(* Prozess Stop *)
IF RisingEdgeProcessStop.Q THEN
	IF NOT(T_Process.T_Ctrle.xDone) AND NOT(T_Process.T_Fct.xExecute) THEN
		(* Prozess muss Aktiv sein und dürfte auch im ZyklusStop Zustand sein, welches dann unterbrochen werden würde *)
		T_Process.T_Fct.xStop:=T_Process.T_Ctrle.xStop;
	ELSE
		T_Process.T_Ctrle.xStop:=FALSE;
	END_IF;
END_IF;
(* Abbrechen des Prozesses *)
IF RisingEdgeProcessAbord.Q THEN
	T_Process.T_Fct.xAbordProcess:=TRUE;
END_IF;
(* Auffangen des Prozess Endes *)
IF NOT(T_Process.T_Ctrle.xDone) AND NOT(T_Process.T_Ctrle.xErrorReady) THEN
	IF NOT(T_Process.T_Fct.xExecute) AND T_Process.T_Fct.xDone THEN
		xSetEnd:=TRUE;
	END_IF;
END_IF;
END_ACTION
ACTION CtrlWorkpiece:
RisingEdgeCheckWorkEnd(CLK:=TStation_Work_St1.THWWorkStation.TCtrlWork.xWorkingFinished);
IF RisingEdgeCheckWorkEnd.Q AND xAutoActiveProcess AND (TStation_Work_St1.THWWorkStation.TCtrlWork.bPartQuality <> 0) AND
     (TStation_Work_St1.THWWorkStation.TCtrlWork.bPartQuality <> 7) AND (TStation_Work_St1.THWWorkStation.TCtrlWork.bPartQuality <> 8) THEN
	(* Nach jeder bearbeitenden Bohrung muss "xAddToolCounter_Machine" gesetzt werden-->Ist für den WzWechsel *)
	TStation_Work_St1.THWWorkStation.TCtrlWork.xAddToolCounter_Machine:=TRUE;
END_IF;
IF xHoleToWork THEN
	IF NOT(xWriteData) THEN
		IF (T_NovRam.T_Parameter.T_PartAnalysis[gciStationSt1].diActual_NumberHoleToWork <= 0) THEN
			T_NovRam.T_Parameter.T_PartAnalysis[gciStationSt1].diActual_NumberHoleToWork:=1;
		END_IF;
		FOR ii:= 1 TO ciMaxWP DO
			IF (T_NovRam.T_Parameter.T_PartAnalysis[gciStationSt1].adiNumberHole[ii] = T_NovRam.T_Parameter.T_PartAnalysis[gciStationSt1].diActual_NumberHoleToWork) THEN
				IF ((T_NovRam.T_Parameter.T_PartAnalysis[gciStationSt1].abWorkPartQuality[ii] >= 1) AND (T_NovRam.T_Parameter.T_PartAnalysis[gciStationSt1].abWorkPartQuality[ii] <= 6)) OR (T_NovRam.T_Parameter.T_PartAnalysis[gciStationSt1].abWorkPartQuality[ii] = 10) THEN
					T_NovRam.T_Parameter.T_PartAnalysis[gciStationSt1].diActual_NumberHoleToWork:=T_NovRam.T_Parameter.T_PartAnalysis[gciStationSt1].diActual_NumberHoleToWork + 1;
				END_IF;
			END_IF;
		END_FOR;
		(* Überprüfe ob Arrayelement erreicht wurde *)
		IF (T_NovRam.T_Parameter.T_PartAnalysis[gciStationSt1].diActual_NumberHoleToWork > T_NovRam.T_Parameter.T_PartAnalysis[gciStationSt1].adiNumberHole[ciMaxWP]) THEN
			FOR ii:=1 TO (ciMaxWP-1) DO
				T_NovRam.T_Parameter.T_PartAnalysis[gciStationSt1].abWorkPartQuality[ii]:=T_NovRam.T_Parameter.T_PartAnalysis[gciStationSt1].abWorkPartQuality[ii+1];
				T_NovRam.T_Parameter.T_PartAnalysis[gciStationSt1].arFirstHC[ii]:=T_NovRam.T_Parameter.T_PartAnalysis[gciStationSt1].arFirstHC[ii+1];
				T_NovRam.T_Parameter.T_PartAnalysis[gciStationSt1].aiHCCounter[ii]:=T_NovRam.T_Parameter.T_PartAnalysis[gciStationSt1].aiHCCounter[ii+1];
				T_NovRam.T_Parameter.T_PartAnalysis[gciStationSt1].aiHCCounterCentering[ii]:=T_NovRam.T_Parameter.T_PartAnalysis[gciStationSt1].aiHCCounterCentering[ii+1];
				T_NovRam.T_Parameter.T_PartAnalysis[gciStationSt1].aiHCCounterTorque[ii]:=T_NovRam.T_Parameter.T_PartAnalysis[gciStationSt1].aiHCCounterTorque[ii+1];
				T_NovRam.T_Parameter.T_PartAnalysis[gciStationSt1].aiHCCounterSpeed[ii]:=T_NovRam.T_Parameter.T_PartAnalysis[gciStationSt1].aiHCCounterSpeed[ii+1];
				T_NovRam.T_Parameter.T_PartAnalysis[gciStationSt1].adiCycleTime[ii]:=T_NovRam.T_Parameter.T_PartAnalysis[gciStationSt1].adiCycleTime[ii+1];
				T_NovRam.T_Parameter.T_PartAnalysis[gciStationSt1].adiWorkTime[ii]:=T_NovRam.T_Parameter.T_PartAnalysis[gciStationSt1].adiWorkTime[ii+1];
				T_NovRam.T_Parameter.T_PartAnalysis[gciStationSt1].abInfeedCounterZ[ii]:=T_NovRam.T_Parameter.T_PartAnalysis[gciStationSt1].abInfeedCounterZ[ii+1];
				T_NovRam.T_Parameter.T_PartAnalysis[gciStationSt1].adiNumberHole[ii]:=T_NovRam.T_Parameter.T_PartAnalysis[gciStationSt1].adiNumberHole[ii+1];
			END_FOR;
			T_NovRam.T_Parameter.T_PartAnalysis[gciStationSt1].abWorkPartQuality[ciMaxWP]:=0;
			T_NovRam.T_Parameter.T_PartAnalysis[gciStationSt1].arFirstHC[ciMaxWP]:=0.0;
			T_NovRam.T_Parameter.T_PartAnalysis[gciStationSt1].aiHCCounter[ciMaxWP]:=0;
			T_NovRam.T_Parameter.T_PartAnalysis[gciStationSt1].aiHCCounterCentering[ciMaxWP]:=0;
			T_NovRam.T_Parameter.T_PartAnalysis[gciStationSt1].aiHCCounterTorque[ciMaxWP]:=0;
			T_NovRam.T_Parameter.T_PartAnalysis[gciStationSt1].aiHCCounterSpeed[ciMaxWP]:=0;
			T_NovRam.T_Parameter.T_PartAnalysis[gciStationSt1].adiCycleTime[ciMaxWP]:=0;
			T_NovRam.T_Parameter.T_PartAnalysis[gciStationSt1].adiWorkTime[ciMaxWP]:=0;
			T_NovRam.T_Parameter.T_PartAnalysis[gciStationSt1].abInfeedCounterZ[ciMaxWP]:=0;
			T_NovRam.T_Parameter.T_PartAnalysis[gciStationSt1].adiNumberHole[ciMaxWP]:=T_NovRam.T_Parameter.T_PartAnalysis[gciStationSt1].adiNumberHole[ciMaxWP] + 1;
		END_IF;
		xHoleToWork:=FALSE;
	END_IF;
END_IF;
END_ACTION
ACTION ProcessFunction_Ctrl_End:
IF T_Process.T_Fct.xSetEndFunction OR xPrcFct_ForceResetFlag THEN
	IF NOT(xPrcFct_ForceResetFlag) THEN
		T_Process.T_Fct.xDone:=TRUE;
	END_IF;
	xPrcFct_ForceResetFlag:=FALSE;
	T_Process.T_Fct.xStop:=FALSE;
	T_Process.T_Fct.xExecute:=FALSE;
	T_Process.T_Fct.xAbordProcess:=FALSE;
	T_Process.T_Fct.xError:=FALSE;
	T_Process.T_Fct.diErrorNr:=0;
	T_Process.T_Fct.xQuitError:=FALSE;
	T_Process.T_Fct.xSetEndFunction:=FALSE;
	T_Process.T_Fct.xReset:=FALSE;
	xPrcFct_SaveStationError:=FALSE;
	xPrcFct_StartPrc_Parallel1:=FALSE;
	xPrcFct_StartPrc_Parallel2:=FALSE;
	iPrcFct_StepPrc_Parallel1:=1;
	iPrcFct_StepPrc_Parallel2:=1;
	xPrcFct_InitStep_Parallel1:=FALSE;
	xPrcFct_InitStep_Parallel2:=FALSE;
	xPrcFct_SetNextStationActive_St1:=FALSE;
	iPrcFct_PickPlaceProcedure:=0;
	xPrcFct_PartDiscReady:=FALSE;
	xPrcFct_ReadyToWriteQuality_St1:=FALSE;
	xPrcFct_XAxisGoToWaitPos:=FALSE;
	xPrcFct_ProcessContinueActive:=FALSE;
	iPrcFct_StepPrc:=1;
	xPrcFct_InitStep:=FALSE;
	xPrcFct_SaveNoMoreParts:=FALSE;
	xPrcFct_StopProcess:=FALSE;
	xPrcFct_StopCycleProcess:=FALSE;
	diPrcFct_SaveErrorNr:=0;
	TStation_Work.THWWorkStation.TCtrlWork.xWP_Analyse_ActiveCycle:=FALSE;			(* Zykluszeit für zu bearbeitende Bohrung ist gestartet *)
	TStation_Work.THWWorkStation.TCtrlWork.xWP_Analyse_ActiveWork:=FALSE;			(* Bearbeitungszeit für zu bearbeitende Bohrung ist gestartet *)
	xStartWorkPart:=FALSE;
	QxCoolant_St1:=FALSE;
	QxFastStrokeOn_St1:=FALSE;
END_IF;
END_ACTION
ACTION ProcessFunction_Ctrl_Error:
xPrcFct_StationError:=	TStation_Work.TControl.xError OR T_ProcessData.T_Ctrle.xErr;
IF (xPrcFct_StationError OR xPrcFct_SaveStationError) AND NOT(T_Process.T_Fct.xErrorReady) THEN
	xPrcFct_SaveStationError:=TRUE;
	IF (T_Process.T_Fct.iFunctNr = 2) THEN
		(* Automat *)
		xPrcFct_WorkStationReady:=	TStation_Work.TControl.xError OR NOT(xStartWorkPart);
	ELSE
		(* Restliche Prozesse *)
		xPrcFct_WorkStationReady:=	(TStation_Work.TControl.xError OR TStation_Work.TControl.xDone);
	END_IF;
	xPrcFct_StationReady:=	(xPrcFct_WorkStationReady OR xPrcFct_StationBlock);
	CASE iPrcFct_StepStationError OF
	(* Abwarten bis alle Station Zyklus beendet haben *)
	1: 	IF xPrcFct_StationReady THEN
			xPrcFct_StationBlock:=TRUE;
			iPrcFct_StepStationError:=iPrcFct_StepStationError + 1;
			IF TStation_Work.THWWorkStation.TCtrlWork.xWorkStartToolRotation THEN
				TStation_Work.THWWorkStation.TCtrlWork.xWorkStopToolRotation:=TRUE;
			END_IF;
		END_IF;
	2:	iPrcFct_StepStationError:=iPrcFct_StepStationError + 1;
		TStation_Work.THWWorkStation.TCtrlWork.xActiveProcess:=FALSE;
		TStation_Work.THWWorkStation.TCtrlWork.xWorkingFinished:=FALSE;
	(* Überprüfen ob es einen Fehler oder eine Warnung ist *)
	3:	IF (diPrcFct_SaveErrorNr <> 0)THEN
			T_Process.T_Fct.diErrorNr:=diPrcFct_SaveErrorNr;
		ELSIF TStation_Work.TControl.xError THEN
			T_Process.T_Fct.diErrorNr:=TStation_Work.TControl.diErrorNr;
		ELSIF T_ProcessData.T_Ctrle.xErr THEN
			T_Process.T_Fct.diErrorNr:=82000000 + T_ProcessData.T_Ctrle.udiErrorID;
		END_IF;
		FBErrorMessage(	diErrorNr:=T_Process.T_Fct.diErrorNr,
							T_ErrorList:=T_ErrorList);
		T_Process.T_Fct.xError:=TRUE;
		diPrcFct_SaveErrorNr:=0;
		iPrcFct_StepStationError:=iPrcFct_StepStationError + 1;
	(* Warten bis Quittiert wird *)
	4:	IF T_Process.T_Fct.xQuitError THEN
			T_Process.T_Fct.xQuitError:=FALSE;
			T_Process.T_Fct.xErrorReady:=TRUE;
			T_Process.T_Fct.xError:=FALSE;
			T_Process.T_Fct.xSetEndFunction:=TRUE;
		END_IF;
	END_CASE;
ELSE
	xExecuteOneTime:=FALSE;
	iPrcFct_StepStationError:=1;
END_IF;
END_ACTION
ACTION ProcessFunction_Ctrl_Main:
(* Prozess Start *)
IF T_Process.T_Fct.xExecute THEN
	T_Process.T_Fct.xStop:=FALSE;
	T_Process.T_Fct.xExecute:=FALSE;
	T_Process.T_Fct.xDone:=FALSE;
	T_Process.T_Fct.xAbordProcess:=FALSE;
	T_Process.T_Fct.xError:=FALSE;
	T_Process.T_Fct.diErrorNr:=0;
	iPrcFct_StepPrc:=1;
	xPrcFct_InitStep:=FALSE;
	xPrcFct_StartMainPrc:=TRUE;
	diPrcFct_SaveErrorNr:=0;
	TStation_Work.THWWorkStation.TCtrlWork.xWorkStartToolRotation:=FALSE;
	TStation_Work.THWWorkStation.TCtrlWork.xWorkStopToolRotation:=FALSE;
	TStation_Work.THWWorkStation.TCtrlWork.xWorkingFinished:=FALSE;
	xPrcFct_SaveNoMoreParts:=FALSE;
	xProcessActive:=FALSE;
END_IF;
(* Abbrechen des Prozesses *)
IF T_Process.T_Fct.xAbordProcess THEN
	T_Process.T_Fct.xAbordProcess:=FALSE;
	T_Process.T_Fct.xSetEndFunction:=TRUE;
END_IF;
IF NOT(xPrcFct_ForceResetFlag) AND xPrcFct_ProcessContinueActive THEN
	xPrcFct_StationBlock:=FALSE;
END_IF;
END_ACTION
ACTION ProcessFunction_Ctrl_Reset:
IF T_Process.T_Fct.xReset THEN
	T_Process.T_Fct.xSetEndFunction:=TRUE;
END_IF;
END_ACTION
ACTION ProcessFunction_Ctrl_Stop:
IF T_Process.T_Fct.xStop OR xPrcFct_StopProcess THEN
	xPrcFct_StationReady:=	NOT(TStation_Work.TControl.xExecute) AND (TStation_Work.TControl.xDone OR TStation_Work.TControl.xError);
	CASE iPrcFct_StepStopProcess OF
	(* Stoppen der Aktiven Stationen *)
	1:	xPrcFct_StationBlock:=TRUE;
		xPrcFct_StopProcess:=TRUE;
		xPrcFct_ProcessContinueActive:=FALSE;
		TStation_Work.TControl.xStop:=NOT(TStation_Work.TControl.xError) AND NOT(TStation_Work.TControl.xDone) AND xEnergyON;
		(* Flag für die WstkAnalyse zurücksetzen *)
		iPrcFct_StepStopProcess:=iPrcFct_StepStopProcess + 1;
	(* Zurücksetzen der Steuerflag für Bearbstationen *)
	2:	IF xPrcFct_StationReady OR xPrcFct_SaveStationError THEN
			iPrcFct_StepStopProcess:=iPrcFct_StepStopProcess + 1;
			TStation_Work.THWWorkStation.TCtrlWork.xActiveProcess:=FALSE;
			TStation_Work.THWWorkStation.TCtrlWork.xWorkingFinished:=FALSE;
			TStation_Work.THWWorkStation.TCtrlWork.xWorkStopToolRotation:=xEnergyON;
			(* Flag für die WstkAnalyse zurücksetzen *)
		END_IF;
	3:	IF (T_Process.T_Ctrle.iFunctNr <> 1) THEN
			TStation_Work.TControl.iFunctNr:=2;			(* Bearbeitungsstation Grundstellung *)
			TStation_Work.TControl.xExecute:=NOT(TStation_Work.TControl.xError) AND xEnergyON;
			IF (TStation_Work.THWWorkStation.TCtrlWork.bPartQuality >= 1) AND (TStation_Work.THWWorkStation.TCtrlWork.bPartQuality <= 6) THEN
				IF T_NovRam.T_Parameter.T_Machine.T_ParamSystem.xDataFileActive AND NOT(T_NovRam.T_Parameter.T_Machine.xEndlessProcessActive) THEN
					(* Prozessdatei wird geschrieben *)
					T_ProcessData.T_Ctrle.iFunction:=1;
					T_ProcessData.T_Ctrle.xExecute:=TRUE;
				END_IF;
			END_IF;
		END_IF;
		iPrcFct_StepStopProcess:=iPrcFct_StepStopProcess + 1;
	4:	IF NOT(TStation_Work.TControl.xExecute) AND (TStation_Work.TControl.xDone OR TStation_Work.TControl.xError) THEN
			iPrcFct_StepStopProcess:=iPrcFct_StepStopProcess + 1;
		END_IF;
	(* Abwarten bis alle Stationen bereit stehen *)
	5:	IF xPrcFct_StationReady OR xPrcFct_SaveStationError THEN
			iPrcFct_StepStopProcess:=iPrcFct_StepStopProcess + 1;
		END_IF;
	6:	xPrcFct_StopProcess:=FALSE;
		T_Process.T_Fct.xStop:=FALSE;
		IF NOT(xPrcFct_SaveStationError) THEN
			T_Process.T_Fct.xAbordProcess:=TRUE;
		END_IF;
	END_CASE;
ELSE
	iPrcFct_StepStopProcess:=1;
END_IF;
END_ACTION
ACTION ProcessFunction_Fct_Automat:
(******************************************************************************************************************************************)
(****************************				           Reset Processfunktion                                            *****************************)
(******************************************************************************************************************************************)
ProcessFunction_Ctrl_Reset;
(******************************************************************************************************************************************)
(****************************			        Processfunktion Fehler Controller                                    *****************************)
(******************************************************************************************************************************************)
ProcessFunction_Ctrl_Error;
(******************************************************************************************************************************************)
(****************************				    Processfunktion Haupt Controller                               *****************************)
(******************************************************************************************************************************************)
ProcessFunction_Ctrl_Main;
(******************************************************************************************************************************************)
(****************************			         Processfunktion sofort Unterbrechung                           *****************************)
(******************************************************************************************************************************************)
ProcessFunction_Ctrl_Stop;
(******************************************************************************************************************************************)
(****************************			             Processfunktion Hauptablauf                                       *****************************)
(******************************************************************************************************************************************)
ProcessFunction_Fct_Automat_Station;
IF xPrcFct_StartMainPrc AND NOT(xPrcFct_StationBlock) AND NOT(T_Process.T_Fct.xSetEndFunction) AND NOT(xPrcFct_SaveStationError) THEN
	CASE iPrcFct_StepPrc OF
	1:	T_ExchgParam.T_Visu.T_Message.iState:=0;
		IF (T_NovRam.T_Parameter.T_StationWork[gciStationSt1].T_ToolCounter.diMaxNumberToolCycle <> 0) AND
		    (T_NovRam.T_Parameter.T_StationWork[gciStationSt1].T_ToolCounter.diToolCycleCounter >= T_NovRam.T_Parameter.T_StationWork[gciStationSt1].T_ToolCounter.diMaxNumberToolCycle) THEN
			TStation_Work.TControl.xError:=TRUE;
			TStation_Work.TControl.xDone:=FALSE;
			TStation_Work.TControl.diErrorNr:=(gciStationSt1 * 1000000) + 16#F101;		(* WzWechsel muss vorgenommen werden *)
			RETURN;
		END_IF;
		IF (garPositionEndProcCalc[1] > T_NovRam.T_Parameter.T_StationWork[gciStationSt1].T_StProcess.rPositionEndProcMaxInc) AND (T_NovRam.T_Parameter.T_StationWork[gciStationSt1].T_StProcess.xPositionEndProcIncOnOff OR gxProcessCylindricalAreaActive) THEN
			TStation_Work.TControl.xError:=TRUE;
			TStation_Work.TControl.xDone:=FALSE;
			TStation_Work.TControl.diErrorNr:=(gciStationSt1 * 1000000) + 17;		(* Z Bearb EndPos Berechn. > Z Bearb EndPos Max *)
			RETURN;
		END_IF;
		IF (garCentringEndProcCalc[1] > T_NovRam.T_Parameter.T_StationWork[gciStationSt1].T_StProcess.rPositionEndProcMaxInc) AND T_NovRam.T_Parameter.T_StationWork[gciStationSt1].T_StProcess.xCentringEndProcIncOnOff THEN
			TStation_Work.TControl.xError:=TRUE;
			TStation_Work.TControl.xDone:=FALSE;
			TStation_Work.TControl.diErrorNr:=(gciStationSt1 * 1000000) + 19;		(* Z ZentrierPos berechn. > Z Bearb EndPos Max *)
			RETURN;
		END_IF;
		IF NOT(xPrcFct_InitStep) THEN
			xPrcFct_InitStep:=TRUE;
			gdiSavePartQuality:=0;
			xHoleToWork:=TRUE;
		END_IF;
		IF NOT(xHoleToWork) THEN
			xPrcFct_InitStep:=FALSE;
			iPrcFct_StepPrc:=iPrcFct_StepPrc + 1;
		END_IF;
	2:	IF NOT(xPrcFct_InitStep) THEN
			xPrcFct_InitStep:=TRUE;
			TStation_Work.TControl.iFunctNr:=2;		(* Bearbeitungsstation Grundstellung *)
			TStation_Work.TControl.xExecute:=TRUE;
			TStation_Work.THWWorkStation.TCtrlWork.xWP_Analyse_ActiveCycle:=TRUE;			(* Zykluszeit für zu bearbeitende Bohrung ist gestartet *)
		END_IF;
		IF NOT(TStation_Work.TControl.xExecute) AND TStation_Work.TControl.xDone THEN
			TStation_Work.THWWorkStation.TCtrlWork.xWorkStartToolRotation:=TRUE;
			xPrcFct_InitStep:=FALSE;
			iPrcFct_StepPrc:=iPrcFct_StepPrc + 1;
		END_IF;
	3:	IF NOT(xPrcFct_InitStep) THEN
			xPrcFct_InitStep:=TRUE;
			xStartWorkPart:=TRUE;
		END_IF;
		IF NOT(xStartWorkPart) THEN
			xPrcFct_InitStep:=FALSE;
			iPrcFct_StepPrc:=90;
		END_IF;
	90:	iPrcFct_StepPrc:=1;
		xPrcFct_InitStep:=FALSE;
		IF NOT(T_NovRam.T_Parameter.T_Machine.xEndlessProcessActive) THEN
			xPrcFct_StartMainPrc:=FALSE;
			T_Process.T_Fct.xSetEndFunction:=TRUE;	(* Prozess beendet *)
		END_IF;
	END_CASE;
END_IF;
(******************************************************************************************************************************************)
(****************************			             Processfunktion Parallelablauf                                       *****************************)
(******************************************************************************************************************************************)
IF NOT(xPrcFct_StationBlock) AND NOT(T_Process.T_Fct.xSetEndFunction) AND NOT(xPrcFct_SaveStationError) THEN
	IF xPrcFct_StartPrc_Parallel1 THEN
		CASE iPrcFct_StepPrc_Parallel1 OF
		1:	iPrcFct_StepPrc_Parallel1:=1;
			xPrcFct_InitStep_Parallel1:=FALSE;
			xPrcFct_StartPrc_Parallel1:=FALSE;
		END_CASE;
	END_IF;
	IF xPrcFct_StartPrc_Parallel2 THEN
		CASE iPrcFct_StepPrc_Parallel2 OF
		1:	iPrcFct_StepPrc_Parallel2:=1;
			xPrcFct_InitStep_Parallel2:=FALSE;
			xPrcFct_StartPrc_Parallel2:=FALSE;
		END_CASE;
	END_IF;
END_IF;
(******************************************************************************************************************************************)
(****************************				     Processfunktion Endprozedur                                    *****************************)
(******************************************************************************************************************************************)
ProcessFunction_Ctrl_End;
END_ACTION
ACTION ProcessFunction_Fct_Automat_Station:
(*********************************************************************************************************************************)
(***********************************			BEARBSTATION RECHTS			***********************************)
(*********************************************************************************************************************************)
IF xStartWorkPart AND NOT(xPrcFct_StationBlock) THEN
	CASE iStepPrc_1 OF
	(* Zuerst überprüfen welche WstkNummer bearbeitet werden muss *)
	1:	iStepPrc_1:=iStepPrc_1 + 1;
		xInitPrc_1:=FALSE;
		xBlockQuality_StR:=FALSE;
		iNumberTryInfeed:=0;
		TStation_Work.THWWorkStation.TCtrlWork.xLastTryInfeed:=FALSE;
	(* .StationFunction_Fct_04_InfeedWorking*)
	2:	IF NOT(xInitPrc_1) THEN
			xInitPrc_1:=TRUE;
			TStation_Work.TControl.iFunctNr:=4;			(* Wz in das Wstk einfädeln *)
			TStation_Work.TControl.xExecute:=TRUE;
			gxSuspensionONOFF:=TRUE;
		END_IF;
		IF NOT(TStation_Work.TControl.xExecute) AND TStation_Work.TControl.xDone THEN
			gxAddInfeedZ:=TRUE;
			IF (TStation_Work.TControl.wStatus <> 99) THEN
				xInitPrc_1:=FALSE;
				iStepPrc_1:=iStepPrc_1 + 1;
				iNumberTryInfeed:=0;
			ELSE
				iNumberTryInfeed:=iNumberTryInfeed + 1;
				IF (iNumberTryInfeed <= T_NovRam.T_Parameter.T_StationWork[gciStationSt1].T_StProcess.iNumberTryInfeed) THEN
					xInitPrc_1:=FALSE;
					iStepPrc_1:=iStepPrc_1;
					IF (iNumberTryInfeed = T_NovRam.T_Parameter.T_StationWork[gciStationSt1].T_StProcess.iNumberTryInfeed) THEN
						TStation_Work.THWWorkStation.TCtrlWork.xLastTryInfeed:=TRUE;
					END_IF;
				ELSE
					(* Anzahl Einfädelversuche erreicht *)
					TStation_Work.THWWorkStation.TCtrlWork.xWorkingFinished:=TRUE;		(* dieses Loch muss als bearbeitet deklariert werden *)
					TStation_Work.THWWorkStation.TCtrlWork.bPartQuality:=5;	(* < NoGo insert fail > *)
					gxSetPartQuality:=TRUE;
					xInitPrc_1:=FALSE;
					iStepPrc_1:=iStepPrc_1 + 3;
					TStation_Work.THWWorkStation.TCtrlWork.xAddWPCounter_Machine_NIO:=TRUE;
					T_NovRam.T_Parameter.T_Machine.T_ParamAutomat.diNumberPartWorked_St1St2:=T_NovRam.T_Parameter.T_Machine.T_ParamAutomat.diNumberPartWorked_St1St2 + 1;
					TStation_Work.THWWorkStation.TCtrlWork.xWorkStopToolRotation:=TRUE;
				END_IF;
			END_IF;
		END_IF;
	(* .StationFunction_Fct_11_Centring *)
	3:	IF NOT(xInitPrc_1) THEN
			xInitPrc_1:=TRUE;
			TStation_Work.TControl.iFunctNr:=11;			(* Zentrieren *)
			TStation_Work.TControl.xExecute:=gxCentringActive OR gxOnlyCentringActive;
		END_IF;
		IF NOT(TStation_Work.TControl.xExecute) AND TStation_Work.TControl.xDone THEN
			IF (TStation_Work.TControl.wStatus <> 99) THEN
				xInitPrc_1:=FALSE;
				IF gxOnlyCentringActive THEN
					TStation_Work.THWWorkStation.TCtrlWork.bPartQuality:=11;	(* < WP Centered > *)
					iStepPrc_1:=iStepPrc_1 + 3;
				ELSE
					iStepPrc_1:=iStepPrc_1 + 1;
				END_IF;
			ELSE
				TStation_Work.THWWorkStation.TCtrlWork.xWorkingFinished:=TRUE;		(* dieses Loch muss als bearbeitet deklariert werden *)
				TStation_Work.THWWorkStation.TCtrlWork.bPartQuality:=10;	(* < NoGo HC Centr. > *)
				gxSetPartQuality:=TRUE;
				xInitPrc_1:=FALSE;
				iStepPrc_1:=iStepPrc_1 + 2;
				TStation_Work.THWWorkStation.TCtrlWork.xAddWPCounter_Machine_NIO:=TRUE;
				T_NovRam.T_Parameter.T_Machine.T_ParamAutomat.diNumberPartWorked_St1St2:=T_NovRam.T_Parameter.T_Machine.T_ParamAutomat.diNumberPartWorked_St1St2 + 1;
				TStation_Work.THWWorkStation.TCtrlWork.xWorkStopToolRotation:=TRUE;
			END_IF;
		END_IF;
	(* .StationFunction_Fct_05_Working *)
	4:	IF NOT(xInitPrc_1) THEN
			xInitPrc_1:=TRUE;
			TStation_Work.TControl.iFunctNr:=5;			(* Wstk bearbeiten *)
			TStation_Work.TControl.xExecute:=TRUE;
			TStation_Work.THWWorkStation.TCtrlWork.xWP_Analyse_ActiveWork:=TRUE;			(* Bearbeitungszeit für zu bearbeitende Bohrung ist gestartet *)
			QxCoolant_St1:=T_NovRam.T_Parameter.T_StationWork[gciStationSt1].T_StProcess.xActivateCoolantProcess;
		END_IF;
		IF TStation_Work.THWWorkStation.TCtrlWork.xWorkingFinished
		AND ((TStation_Work.THWWorkStation.TAxisZ.T_LiveValue.lrActualPosition <= T_NovRam.T_Parameter.T_StationWork[gciStationSt1].T_StProcess.rStrokeAxisPosSwitchCoolantOff)
		OR (TStation_Work.THWWorkStation.TAxisZ.T_LiveValue.lrActualPosition <= T_NovRam.T_Parameter.T_StationWork[gciStationSt1].T_StProcess.rPositionStartProc)) THEN
			QxCoolant_St1:=FALSE;
		END_IF;
		IF TStation_Work.THWWorkStation.TCtrlWork.xWorkingFinished AND NOT(xBlockQuality_StR) THEN
			xBlockQuality_StR:=TRUE;
			IF (TStation_Work.THWWorkStation.TCtrlWork.bPartQuality = 1) OR (TStation_Work.THWWorkStation.TCtrlWork.bPartQuality = 2) THEN
				TStation_Work.THWWorkStation.TCtrlWork.xAddWPCounter_Machine_IO:=TRUE;
				T_NovRam.T_Parameter.T_Machine.T_ParamAutomat.diNumberPartWorked_St1St2:=T_NovRam.T_Parameter.T_Machine.T_ParamAutomat.diNumberPartWorked_St1St2 + 1;
			ELSIF (TStation_Work.THWWorkStation.TCtrlWork.bPartQuality <> 7) AND (TStation_Work.THWWorkStation.TCtrlWork.bPartQuality <> 8) THEN
				TStation_Work.THWWorkStation.TCtrlWork.xAddWPCounter_Machine_NIO:=TRUE;
				T_NovRam.T_Parameter.T_Machine.T_ParamAutomat.diNumberPartWorked_St1St2:=T_NovRam.T_Parameter.T_Machine.T_ParamAutomat.diNumberPartWorked_St1St2 + 1;
			END_IF;
		END_IF;
		IF NOT(TStation_Work.TControl.xExecute) AND TStation_Work.TControl.xDone THEN
			xBlockQuality_StR:=FALSE;
			iStepPrc_1:=iStepPrc_1 + 1;
			xInitPrc_1:=FALSE;
		END_IF;
	5:	IF NOT(xInitPrc_1) THEN
			xInitPrc_1:=TRUE;
			IF T_NovRam.T_Parameter.T_Machine.T_ParamSystem.xDataFileActive AND NOT(T_NovRam.T_Parameter.T_Machine.xEndlessProcessActive) THEN
				(* Prozessdatei wird geschrieben *)
				T_ProcessData.T_Ctrle.iFunction:=1;
				T_ProcessData.T_Ctrle.xExecute:=TRUE;
			END_IF;
		END_IF;
		IF NOT(T_ProcessData.T_Ctrle.xExecute) AND T_ProcessData.T_Ctrle.xDone THEN
			iStepPrc_1:=iStepPrc_1 + 1;
			xInitPrc_1:=FALSE;
		END_IF;
		IF T_ProcessData.T_Ctrle.xErr THEN
			xStartWorkPart:=FALSE;
		END_IF;
	6:	IF NOT(xInitPrc_1) THEN
			xInitPrc_1:=TRUE;
			gxSuspensionONOFF:=FALSE;
		END_IF;
		IF TRUE THEN
			iStepPrc_1:=1;
			xInitPrc_1:=FALSE;
			TStation_Work.THWWorkStation.TCtrlWork.xWP_Analyse_ActiveCycle:=FALSE;			(* Zykluszeit für zu bearbeitende Bohrung ist gestoppt *)
			xStartWorkPart:=FALSE;
		END_IF;
	END_CASE;
ELSE
	iStepPrc_1:=1;
	xInitPrc_1:=FALSE;
END_IF;
END_ACTION
ACTION ProcessFunction_Fct_HandMode:
(******************************************************************************************************************************************)
(****************************				           Reset Processfunktion                                            *****************************)
(******************************************************************************************************************************************)
ProcessFunction_Ctrl_Reset;
(******************************************************************************************************************************************)
(****************************			        Processfunktion Fehler Controller                                    *****************************)
(******************************************************************************************************************************************)
ProcessFunction_Ctrl_Error;
(******************************************************************************************************************************************)
(****************************				    Processfunktion Haupt Controller                               *****************************)
(******************************************************************************************************************************************)
ProcessFunction_Ctrl_Main;
(******************************************************************************************************************************************)
(****************************			         Processfunktion sofort Unterbrechung                           *****************************)
(******************************************************************************************************************************************)
ProcessFunction_Ctrl_Stop;
(******************************************************************************************************************************************)
(****************************			             Processfunktion Hauptablauf                                       *****************************)
(******************************************************************************************************************************************)
ProcessFunction_Fct_Automat_Station;
IF xPrcFct_StartMainPrc AND NOT(xPrcFct_StationBlock) AND NOT(T_Process.T_Fct.xSetEndFunction) AND NOT(xPrcFct_SaveStationError) THEN
	CASE iPrcFct_StepPrc OF
	(* Grundstellung *)
	1:	IF (garPositionEndProcCalc[1] > T_NovRam.T_Parameter.T_StationWork[gciStationSt1].T_StProcess.rPositionEndProcMaxInc) AND (T_NovRam.T_Parameter.T_StationWork[gciStationSt1].T_StProcess.xPositionEndProcIncOnOff OR gxProcessCylindricalAreaActive) THEN
			TStation_Work.TControl.xError:=TRUE;
			TStation_Work.TControl.xDone:=FALSE;
			TStation_Work.TControl.diErrorNr:=(gciStationSt1 * 1000000) + 17;		(* Z Bearb EndPos Berechn. > Z Bearb EndPos Max *)
			RETURN;
		END_IF;
		IF (garCentringEndProcCalc[1] > T_NovRam.T_Parameter.T_StationWork[gciStationSt1].T_StProcess.rPositionEndProcMaxInc) AND T_NovRam.T_Parameter.T_StationWork[gciStationSt1].T_StProcess.xCentringEndProcIncOnOff THEN
			TStation_Work.TControl.xError:=TRUE;
			TStation_Work.TControl.xDone:=FALSE;
			TStation_Work.TControl.diErrorNr:=(gciStationSt1 * 1000000) + 19;		(* Z ZentrierPos berechn. > Z Bearb EndPos Max *)
			RETURN;
		END_IF;
		IF NOT(xPrcFct_InitStep) THEN
			xPrcFct_InitStep:=TRUE;
			TStation_Work.TControl.iFunctNr:=2;		(* Bearbeitungsstation Grundstellung *)
			TStation_Work.TControl.xExecute:=TRUE;
			iNumberTryInfeed:=0;
			TStation_Work.THWWorkStation.TCtrlWork.xWP_Analyse_ActiveCycle:=TRUE;			(* Zykluszeit für zu bearbeitende Bohrung ist gestartet *)
			gxSuspensionONOFF:=TRUE;
		END_IF;
		IF NOT(TStation_Work.TControl.xExecute) AND TStation_Work.TControl.xDone THEN
			TStation_Work.THWWorkStation.TCtrlWork.xWorkStartToolRotation:=TRUE;
			xPrcFct_InitStep:=FALSE;
			iPrcFct_StepPrc:=iPrcFct_StepPrc + 1;
			TStation_Work.THWWorkStation.TCtrlWork.xLastTryInfeed:=FALSE;
		END_IF;
	(* Wz in das Wstk einfädeln *)
	2:	IF NOT(xPrcFct_InitStep) THEN
			xPrcFct_InitStep:=TRUE;
			TStation_Work.TControl.iFunctNr:=4;		(* Wz Einfädeln *)
			TStation_Work.TControl.xExecute:=TRUE;
		END_IF;
		IF NOT(TStation_Work.TControl.xExecute) AND TStation_Work.TControl.xDone THEN
			IF (TStation_Work.TControl.wStatus <> 99) THEN
				xPrcFct_InitStep:=FALSE;
				iPrcFct_StepPrc:=iPrcFct_StepPrc + 1;
			ELSE
				iNumberTryInfeed:=iNumberTryInfeed + 1;
				IF (iNumberTryInfeed <= T_NovRam.T_Parameter.T_StationWork[gciStationSt1].T_StProcess.iNumberTryInfeed) THEN
					xPrcFct_InitStep:=FALSE;
					iPrcFct_StepPrc:=iPrcFct_StepPrc;
					IF (iNumberTryInfeed = T_NovRam.T_Parameter.T_StationWork[gciStationSt1].T_StProcess.iNumberTryInfeed) THEN
						TStation_Work.THWWorkStation.TCtrlWork.xLastTryInfeed:=TRUE;
					END_IF;
				ELSE
					(* Anzahl Einfädelversuche erreicht *)
					TStation_Work.THWWorkStation.TCtrlWork.bPartQuality:=5;	(* < NoGo insert fail > *)
					TStation_Work.THWWorkStation.TCtrlWork.xWP_Analyse_ActiveWork:=FALSE;
					TStation_Work.THWWorkStation.TCtrlWork.xWorkStopToolRotation:=TRUE;
					TStation_Work.THWWorkStation.TCtrlWork.xWorkingFinished:=TRUE;
					xPrcFct_InitStep:=FALSE;
					iPrcFct_StepPrc:=iPrcFct_StepPrc + 3;
				END_IF;
			END_IF;
		END_IF;



	(* .StationFunction_Fct_11_Centring *)
	3:	IF NOT(xPrcFct_InitStep) THEN
			xPrcFct_InitStep:=TRUE;
			TStation_Work.TControl.iFunctNr:=11;			(* Zentrieren *)
			TStation_Work.TControl.xExecute:=gxCentringActive OR gxOnlyCentringActive;
		END_IF;
		IF NOT(TStation_Work.TControl.xExecute) AND TStation_Work.TControl.xDone THEN
			IF (TStation_Work.TControl.wStatus <> 99) THEN
				xPrcFct_InitStep:=FALSE;
				IF gxOnlyCentringActive THEN
					TStation_Work.THWWorkStation.TCtrlWork.bPartQuality:=11;	(* < WP Centered > *)
					iPrcFct_StepPrc:=iPrcFct_StepPrc + 2;
				ELSE
					iPrcFct_StepPrc:=iPrcFct_StepPrc + 1;
				END_IF;
			ELSE
				TStation_Work.THWWorkStation.TCtrlWork.bPartQuality:=10;	(* < NoGo HC Centr. > *)
				xPrcFct_InitStep:=FALSE;
				iPrcFct_StepPrc:=iPrcFct_StepPrc + 2;
				TStation_Work.THWWorkStation.TCtrlWork.xAddWPCounter_Machine_NIO:=TRUE;
				T_NovRam.T_Parameter.T_Machine.T_ParamAutomat.diNumberPartWorked_St1St2:=T_NovRam.T_Parameter.T_Machine.T_ParamAutomat.diNumberPartWorked_St1St2 + 1;
				TStation_Work.THWWorkStation.TCtrlWork.xWorkStopToolRotation:=TRUE;
			END_IF;
		END_IF;



	(* Wstk bearbeiten *)
	4:	IF NOT(xPrcFct_InitStep) THEN
			xPrcFct_InitStep:=TRUE;
			TStation_Work.TControl.iFunctNr:=5;		(* Wstk bearbeiten *)
			TStation_Work.TControl.xExecute:=TRUE;
			TStation_Work.THWWorkStation.TCtrlWork.xWP_Analyse_ActiveWork:=TRUE;			(* Bearbeitungszeit für zu bearbeitende Bohrung ist gestartet *)
			QxCoolant_St1:=T_NovRam.T_Parameter.T_StationWork[gciStationSt1].T_StProcess.xActivateCoolantProcess;
		END_IF;
		IF TStation_Work.THWWorkStation.TCtrlWork.xWorkingFinished
		AND ((TStation_Work.THWWorkStation.TAxisZ.T_LiveValue.lrActualPosition <= T_NovRam.T_Parameter.T_StationWork[gciStationSt1].T_StProcess.rStrokeAxisPosSwitchCoolantOff)
		OR (TStation_Work.THWWorkStation.TAxisZ.T_LiveValue.lrActualPosition <= T_NovRam.T_Parameter.T_StationWork[gciStationSt1].T_StProcess.rPositionStartProc)) THEN
			QxCoolant_St1:=FALSE;
		END_IF;
		IF NOT(TStation_Work.TControl.xExecute) AND TStation_Work.TControl.xDone THEN
			xPrcFct_InitStep:=FALSE;
			iPrcFct_StepPrc:=iPrcFct_StepPrc + 1;
			xActivate_StationRight:=FALSE;
			TStation_Work.THWWorkStation.TCtrlWork.xWorkStopToolRotation:=TRUE;
		END_IF;
		IF TStation_Work.THWWorkStation.TCtrlWork.xWorkingFinished THEN
			IF (TStation_Work.THWWorkStation.TCtrlWork.bPartQuality <> 0) AND (TStation_Work.THWWorkStation.TCtrlWork.bPartQuality <> 7) AND
			     (TStation_Work.THWWorkStation.TCtrlWork.bPartQuality <> 8) THEN
				TStation_Work.THWWorkStation.TCtrlWork.xWP_Analyse_ActiveWork:=FALSE;			(* Bearbeitungszeit für zu bearbeitende Bohrung ist gestoppt *)
			END_IF;
		END_IF;
	(* Grundstellung *)
	5:	IF NOT(xPrcFct_InitStep) THEN
			xPrcFct_InitStep:=TRUE;
			TStation_Work.TControl.iFunctNr:=2;		(* BearbeitStation Grundstellung *)
			TStation_Work.TControl.xExecute:=TRUE;
			gxBlockSetQuality:=TRUE;
		END_IF;
		IF NOT(TStation_Work.TControl.xExecute) AND TStation_Work.TControl.xDone THEN
			TStation_Work.THWWorkStation.TCtrlWork.xWP_Analyse_ActiveCycle:=FALSE;			(* Zykluszeit für zu bearbeitende Bohrung ist gestoppt *)
			gxWP_Analyse_ActiveWork:=FALSE;
			gxWP_Analyse_ActiveWork:=FALSE;
			xPrcFct_InitStep:=FALSE;
			iPrcFct_StepPrc:=90;
		END_IF;



	(* Ende HandBetrieb Prozess *)
	90:	iPrcFct_StepPrc:=1;
		xPrcFct_InitStep:=FALSE;
		xPrcFct_StartMainPrc:=FALSE;
		T_Process.T_Fct.xSetEndFunction:=TRUE;	(* Prozess beendet *)
		gxSuspensionONOFF:=FALSE;
	END_CASE;
END_IF;
(******************************************************************************************************************************************)
(****************************			             Processfunktion Parallelablauf                                       *****************************)
(******************************************************************************************************************************************)

(******************************************************************************************************************************************)
(****************************				     Processfunktion Endprozedur                                    *****************************)
(******************************************************************************************************************************************)
ProcessFunction_Ctrl_End;
END_ACTION
ACTION ProcessFunction_Fct_Referencing:
(******************************************************************************************************************************************)
(****************************				           Reset Processfunktion                                            *****************************)
(******************************************************************************************************************************************)
ProcessFunction_Ctrl_Reset;
(******************************************************************************************************************************************)
(****************************			        Processfunktion Fehler Controller                                    *****************************)
(******************************************************************************************************************************************)
ProcessFunction_Ctrl_Error;
(******************************************************************************************************************************************)
(****************************				    Processfunktion Haupt Controller                               *****************************)
(******************************************************************************************************************************************)
ProcessFunction_Ctrl_Main;
(******************************************************************************************************************************************)
(****************************			         Processfunktion sofort Unterbrechung                           *****************************)
(******************************************************************************************************************************************)
ProcessFunction_Ctrl_Stop;
(******************************************************************************************************************************************)
(****************************			             Processfunktion Hauptablauf                                       *****************************)
(******************************************************************************************************************************************)
IF xPrcFct_StartMainPrc AND NOT(xPrcFct_StationBlock) AND NOT(T_Process.T_Fct.xSetEndFunction) AND NOT(xPrcFct_SaveStationError) THEN
	CASE iPrcFct_StepPrc OF
	1:	gxInitialStateActivated:=FALSE;
		xSpindelCalibrationONOFF:=gxSpindelCalibrationONOFF_St1;
		xPrcFct_Ready_St1:=FALSE;
		xPrcFct_InitStep:=FALSE;
		iPrcFct_StepPrc:=iPrcFct_StepPrc + 1;
	2:	IF NOT(xPrcFct_InitStep) THEN
			xPrcFct_InitStep:=TRUE;
			xPrcFct_StartPrc_Parallel1:=TRUE;
		END_IF;
		IF xPrcFct_Ready_St1 THEN
			xPrcFct_InitStep:=FALSE;
			iPrcFct_StepPrc:=iPrcFct_StepPrc + 1;
		END_IF;
	3:	IF NOT(xPrcFct_StartPrc_Parallel1) THEN
			gxInitialStateActivated:=TRUE;
			iPrcFct_StepPrc:=1;
			xPrcFct_InitStep:=FALSE;
			xPrcFct_StartMainPrc:=FALSE;
			T_Process.T_Fct.xSetEndFunction:=TRUE;
		END_IF;
	END_CASE;
END_IF;
(******************************************************************************************************************************************)
(****************************			             Processfunktion Parallelablauf                                       *****************************)
(******************************************************************************************************************************************)
IF NOT(xPrcFct_StationBlock) AND NOT(T_Process.T_Fct.xSetEndFunction) AND NOT(xPrcFct_SaveStationError) THEN
	IF xPrcFct_StartPrc_Parallel1 THEN
		CASE iPrcFct_StepPrc_Parallel1 OF
		1:	IF NOT(xPrcFct_InitStep_Parallel1) THEN
				xPrcFct_InitStep_Parallel1:=TRUE;
				TStation_Work.TControl.iFunctNr:=2;	(* Bearbeitungsstation Grundstellung *)
				TStation_Work.TControl.xExecute:=TRUE;
			END_IF;
			IF NOT(TStation_Work.TControl.xExecute) AND TStation_Work.TControl.xDone THEN
				iPrcFct_StepPrc_Parallel1:=iPrcFct_StepPrc_Parallel1 + 1;
				xPrcFct_InitStep_Parallel1:=FALSE;
			END_IF;
		2:	IF NOT(xPrcFct_InitStep_Parallel1) THEN
				xPrcFct_InitStep_Parallel1:=TRUE;
				TStation_Work.TControl.iFunctNr:=10;	(* Überprüfen ob die Achsenbremse blockiert ist, damit im Fall dass sie blockiert ist eine Vorwarnung ausgegeben werden kann *)
				TStation_Work.TControl.xExecute:=TRUE;
				xPrcFct_Ready_St1:=TRUE;
			END_IF;
			IF NOT(TStation_Work.TControl.xExecute) AND TStation_Work.TControl.xDone THEN
				iPrcFct_StepPrc_Parallel1:=iPrcFct_StepPrc_Parallel1 + 1;
				xPrcFct_InitStep_Parallel1:=FALSE;
			END_IF;
		3:	IF NOT(xPrcFct_InitStep_Parallel1) THEN
				xPrcFct_InitStep_Parallel1:=TRUE;
				(* Existierende MicroHead Bearbstationen müssen noch kalibriert werden *)
				TStation_Work.TControl.iFunctNr:=7;		(* Kalibrierung starten *)
				TStation_Work.THWWorkStation.TCtrlWork.xActiveCalibrateToolDeflection:=xSpindelCalibrationONOFF;
				TStation_Work.THWWorkStation.TCtrlWork.xActiveCalibrateToolTorque:=xSpindelCalibrationONOFF;
				TStation_Work.THWWorkStation.TCtrlWork.xStopToolRotation:=xSpindelCalibrationONOFF;
				TStation_Work.TControl.xExecute:=xSpindelCalibrationONOFF;
			END_IF;
			IF ((NOT(TStation_Work.TControl.xExecute) AND TStation_Work.TControl.xDone AND xSpindelCalibrationONOFF) OR NOT(xSpindelCalibrationONOFF)) THEN
				iPrcFct_StepPrc_Parallel1:=1;
				xPrcFct_InitStep_Parallel1:=FALSE;
				xPrcFct_StartPrc_Parallel1:=FALSE;
			END_IF;
		END_CASE;
	END_IF;
ELSE
	iPrcFct_StepPrc_Parallel1:=1;
	xPrcFct_InitStep_Parallel1:=FALSE;
END_IF;
(******************************************************************************************************************************************)
(****************************				     Processfunktion Endprozedur                                    *****************************)
(******************************************************************************************************************************************)
ProcessFunction_Ctrl_End;
END_ACTION

(* POU PRG_LAYER4_PROCESS/FBPROCESS/FB_ProcessInformation, ST *)
FUNCTION_BLOCK FB_ProcessInformation
VAR_INPUT
END_VAR
VAR_IN_OUT
	T_Parameter:ST_RETAIN_DATA;
	TStation_Work : ST_STATION;
END_VAR
VAR_OUTPUT
END_VAR
VAR
	TONWorkTime: TON;
	TONCycleTime: TON;
	RisingEdgeStartWorkProcess: R_TRIG;
	RisingEdgeStartCycleProcess: R_TRIG;
	RisingEdgeStationFunction: R_TRIG;
END_VAR
RisingEdgeStartCycleProcess(CLK:=TStation_Work.THWWorkStation.TCtrlWork.xWP_Analyse_ActiveCycle);
RisingEdgeStartWorkProcess(CLK:=TStation_Work.THWWorkStation.TCtrlWork.xWP_Analyse_ActiveWork);
RisingEdgeStationFunction(CLK:=gxWP_Analyse_ActiveWork);

IF TStation_Work.THWWorkStation.TCtrlWork.xWP_Analyse_ActiveCycle THEN
	IF RisingEdgeStartCycleProcess.Q THEN
		T_Parameter.T_StationWork[gciStationSt1].T_InfoProcess.tLastCycleTime:=T_Parameter.T_StationWork[gciStationSt1].T_InfoProcess.tActualCycleTime;
		T_Parameter.T_StationWork[gciStationSt1].T_InfoProcess.tActualCycleTime:=T#0s;
		T_Parameter.T_StationWork[gciStationSt1].T_InfoProcess.rActualCycleTime:=0.0;
		TONCycleTime(IN:=FALSE);
	END_IF;
	TONCycleTime(IN:=TRUE,PT:=T#999999s);
	T_Parameter.T_StationWork[gciStationSt1].T_InfoProcess.tActualCycleTime:=TONCycleTime.ET;
	T_Parameter.T_StationWork[gciStationSt1].T_InfoProcess.rActualCycleTime:=TIME_TO_REAL(TONCycleTime.ET)/1000.0;
END_IF;
IF TStation_Work.THWWorkStation.TCtrlWork.xWP_Analyse_ActiveWork OR gxWP_Analyse_ActiveWork THEN
	IF RisingEdgeStartWorkProcess.Q OR RisingEdgeStationFunction.Q THEN
		T_Parameter.T_StationWork[gciStationSt1].T_InfoProcess.tLastEffProcTime:=T_Parameter.T_StationWork[gciStationSt1].T_InfoProcess.tActualEffProcTime;
		T_Parameter.T_StationWork[gciStationSt1].T_InfoProcess.tActualEffProcTime:=T#0s;
		T_Parameter.T_StationWork[gciStationSt1].T_InfoProcess.rActualEffProcTime:=0.0;
		TStation_Work.THWWorkStation.TCtrlWork.rDiffOverLimitPosition:=0.0;
		TONWorkTime(IN:=FALSE);
	END_IF;
	TONWorkTime(IN:=TRUE,PT:=T#999999s);
	T_Parameter.T_StationWork[gciStationSt1].T_InfoProcess.tActualEffProcTime:=TONWorkTime.ET;
	T_Parameter.T_StationWork[gciStationSt1].T_InfoProcess.rActualEffProcTime:=TIME_TO_REAL(TONWorkTime.ET)/1000.0;
END_IF;
IF TStation_Work.THWWorkStation.TCtrlWork.xWP_Analyse_ActiveCycle OR TStation_Work.THWWorkStation.TCtrlWork.xWP_Analyse_ActiveWork OR gxWP_Analyse_ActiveWork THEN
	T_Parameter.T_StationWork[gciStationSt1].T_InfoProcess.rActualFirstContactPosition:=TStation_Work.THWWorkStation.TCtrlWork.rActualFirstContactPosition;
	T_Parameter.T_StationWork[gciStationSt1].T_InfoProcess.rLastFirstContactPosition:=TStation_Work.THWWorkStation.TCtrlWork.rLastFirstContactPosition;
	T_Parameter.T_StationWork[gciStationSt1].T_InfoProcess.rLastOverLimitPosition:=TStation_Work.THWWorkStation.TCtrlWork.rLastOverLimitPosition;
	T_Parameter.T_StationWork[gciStationSt1].T_InfoProcess.rDiffOverLimitPosition:=TStation_Work.THWWorkStation.TCtrlWork.rDiffOverLimitPosition;
	T_Parameter.T_StationWork[gciStationSt1].T_InfoProcess.rCuttingSpeed:=TStation_Work.THWWorkStation.TCtrlWork.rCuttingSpeed;
	T_Parameter.T_StationWork[gciStationSt1].T_InfoProcess.iOverLimitCounter:=TStation_Work.THWWorkStation.TCtrlWork.iOverLimitCounter;

	T_Parameter.T_StationWork[gciStationSt1].T_InfoProcess.iOverLimitCounterCentering:=TStation_Work.THWWorkStation.TCtrlWork.iOverLimitCounterCentering;

	T_Parameter.T_StationWork[gciStationSt1].T_InfoProcess.iOverLimitCounterTorque:=TStation_Work.THWWorkStation.TCtrlWork.iOverLimitCounterTorque;
	T_Parameter.T_StationWork[gciStationSt1].T_InfoProcess.iOverLimitCounterSpeed:=TStation_Work.THWWorkStation.TCtrlWork.iOverLimitCounterSpeed;
	T_Parameter.T_StationWork[gciStationSt1].T_InfoProcess.bLastDetectionSignal:=WORD_TO_BYTE(TStation_Work.TControl.wStatus);
	T_Parameter.T_StationWork[gciStationSt1].T_InfoProcess.bPartQuality:=TStation_Work.THWWorkStation.TCtrlWork.bPartQuality;
	T_Parameter.T_StationWork[gciStationSt1].T_InfoProcess.rProcessWork:=TStation_Work.THWWorkStation.TCtrlWork.rProcessWork;

	T_Parameter.T_StationWork[TStation_Work.iStationNr].T_InfoProcess.rTorqueHC:=TStation_Work.THWWorkStation.TCtrlWork.rTorqueHC;
	T_Parameter.T_StationWork[TStation_Work.iStationNr].T_InfoProcess.rTorqueAfterHC_Min:=TStation_Work.THWWorkStation.TCtrlWork.rTorqueAfterHC_Min;
	T_Parameter.T_StationWork[TStation_Work.iStationNr].T_InfoProcess.rTorqueAfterHC_Max:=TStation_Work.THWWorkStation.TCtrlWork.rTorqueAfterHC_Max;
	T_Parameter.T_StationWork[TStation_Work.iStationNr].T_InfoProcess.xTorqueLastHC:=TStation_Work.THWWorkStation.TCtrlWork.xTorqueLastHC;
	T_Parameter.T_StationWork[TStation_Work.iStationNr].T_InfoProcess.xDeflectionLastHC:=TStation_Work.THWWorkStation.TCtrlWork.xDeflectionLastHC;
	T_Parameter.T_StationWork[TStation_Work.iStationNr].T_InfoProcess.iHCTorquePos:=TStation_Work.THWWorkStation.TCtrlWork.iHCTorquePos;
	T_Parameter.T_StationWork[TStation_Work.iStationNr].T_InfoProcess.iHCDeflectionPos:=TStation_Work.THWWorkStation.TCtrlWork.iHCDeflectionPos;
	T_Parameter.T_StationWork[TStation_Work.iStationNr].T_InfoProcess.xHCSparkOut:=TStation_Work.THWWorkStation.TCtrlWork.xHCSparkOut;
END_IF;
IF gxWP_Analyse_ActiveInfeed THEN
	T_Parameter.T_StationWork[gciStationSt1].T_InfoProcess.bPartQuality:=TStation_Work.THWWorkStation.TCtrlWork.bPartQuality;
END_IF;
IF gxWP_Analyse_ResetCentCountValue THEN
	gxWP_Analyse_ResetCentCountValue:=FALSE;
	T_Parameter.T_StationWork[gciStationSt1].T_InfoProcess.iOverLimitCounterCentering:=TStation_Work.THWWorkStation.TCtrlWork.iOverLimitCounterCentering;
END_IF;
END_FUNCTION_BLOCK

(* POU PRG_LAYER4_PROCESS/FBPROCESS/FB_WPCounter, ST *)
FUNCTION_BLOCK FB_WPCounter
VAR_INPUT
	iStationNr:INT;
END_VAR
VAR_IN_OUT
	T_Parameter:ST_RETAIN_DATA;
	T_CtrlWork:ST_CTRL_WORK;
END_VAR
VAR_OUTPUT
END_VAR
VAR
END_VAR
IF T_CtrlWork.xAddWPCounter_Machine_IO THEN
	T_CtrlWork.xAddWPCounter_Machine_IO:=FALSE;
	T_Parameter.T_StationWork[gciStationSt1].T_WPCounter.diWPCounter_IO_Actual:=
						T_Parameter.T_StationWork[gciStationSt1].T_WPCounter.diWPCounter_IO_Actual + 1;		(* Maschinen Wstk Zähler IO Tagesaktuell nicht rücksetzbar *)
	T_Parameter.T_StationWork[gciStationSt1].T_WPCounter.diWPCounter_IO_Reset:=
						T_Parameter.T_StationWork[gciStationSt1].T_WPCounter.diWPCounter_IO_Reset + 1;		(* Maschinen Wstk Zähler IO Rücksetzbar *)
END_IF;
IF T_CtrlWork.xAddWPCounter_Machine_NIO THEN
	T_CtrlWork.xAddWPCounter_Machine_NIO:=FALSE;
	T_Parameter.T_StationWork[gciStationSt1].T_WPCounter.diWPCounter_NIO_Actual:=
						T_Parameter.T_StationWork[gciStationSt1].T_WPCounter.diWPCounter_NIO_Actual + 1;		(* Maschinen Wstk Zähler NIO Tagesaktuell nicht rücksetzbar *)
	T_Parameter.T_StationWork[gciStationSt1].T_WPCounter.diWPCounter_NIO_Reset:=
						T_Parameter.T_StationWork[gciStationSt1].T_WPCounter.diWPCounter_NIO_Reset + 1;		(* Maschinen Wstk Zähler NIO Rücksetzbar *)
END_IF;

T_Parameter.T_StationWork[gciStationSt1].T_WPCounter.diWPCounter_IO_NIO:=		T_Parameter.T_StationWork[gciStationSt1].T_WPCounter.diWPCounter_IO_Actual +
																				T_Parameter.T_StationWork[gciStationSt1].T_WPCounter.diWPCounter_NIO_Actual;

IF T_CtrlWork.xAddToolCounter_Machine THEN
	T_CtrlWork.xAddToolCounter_Machine:=FALSE;
	IF (T_CtrlWork.bPartQuality >= 1) AND (T_CtrlWork.bPartQuality <= 5) AND NOT(T_NovRam.T_Parameter.T_Machine.xEndlessProcessActive) THEN
		T_Parameter.T_StationWork[gciStationSt1].T_ToolCounter.diToolCycleCounter:=T_Parameter.T_StationWork[gciStationSt1].T_ToolCounter.diToolCycleCounter + 1;	(* Station 1 Wz Zähler um 1 erhöhen *)
	END_IF;
END_IF;
END_FUNCTION_BLOCK

(* POU PRG_LAYER4_PROCESS/FBPROCESS/FB_WPAnalysis, ST *)
FUNCTION_BLOCK FB_WPAnalysis
VAR_INPUT
	diActual_NumberHoleToWork:DINT;		(* Aktuell zu bearbeitende Bohrungsnummer *)
END_VAR
VAR_IN_OUT
	T_PartAnalysis:ST_PARTANALYSIS;
	TStation_Work : ST_STATION;
	xAddInfeedZ:BOOL;
	xSetPartQuality:BOOL;
END_VAR
VAR_OUTPUT
END_VAR
VAR
	TONCycleTime: TON;
	TONWorkTime: TON;
	FBNT_GetTime:NT_GetTime;
	iSetTimeStamp_Start: INT;
	iSetTimeStamp_End: INT;
	diHoleNumber: DINT;
	xInitCycleTime: BOOL;
	tSaveCycleTime: TIME;
	xInitWorkTime: BOOL;
	tSaveWorkTime: TIME;
	ii: INT;
	iHCCounter_Save: INT;
	iHCCounterCentering_Save: INT;
	iHCCounterTorque_Save: INT;
	iHCCounterSpeed_Save:INT;	(* IGS *)
END_VAR
(* Aufzeichnung für wenn die Bearb Station aktiviert wurde *)
IF TStation_Work.THWWorkStation.TCtrlWork.xWP_Analyse_StartAutomat THEN
	CASE iSetTimeStamp_Start OF
	1:	FBNT_GetTime(	NETID:= '',
						START:=FALSE );
		iSetTimeStamp_Start:=iSetTimeStamp_Start + 1;
	2:	FBNT_GetTime(	NETID:= '',
						START:= TRUE,
						TMOUT:= T#2s);
		IF NOT(FBNT_GetTime.BUSY) OR FBNT_GetTime.ERR THEN
			IF NOT(FBNT_GetTime.ERR) THEN
				T_PartAnalysis.sStartOfProcess:=Fct_ConvertDateToString(3,FBNT_GetTime.TIMESTR);
			END_IF;
			iSetTimeStamp_Start:=1;
			TStation_Work.THWWorkStation.TCtrlWork.xWP_Analyse_StartAutomat:=FALSE;
		END_IF;
	END_CASE;
ELSE
	iSetTimeStamp_Start:=1;
END_IF;
IF TStation_Work.THWWorkStation.TCtrlWork.xWP_Analyse_StopAutomat THEN
	CASE iSetTimeStamp_End OF
	1:	FBNT_GetTime(	NETID:= '',
						START:=FALSE );
		iSetTimeStamp_End:=iSetTimeStamp_End + 1;
	2:	FBNT_GetTime(	NETID:= '',
						START:= TRUE,
						TMOUT:= T#2s);
		IF NOT(FBNT_GetTime.BUSY) OR FBNT_GetTime.ERR THEN
			IF NOT(FBNT_GetTime.ERR) THEN
				T_PartAnalysis.sEndOfProcess:=Fct_ConvertDateToString(3,FBNT_GetTime.TIMESTR);
			END_IF;
			iSetTimeStamp_End:=1;
			TStation_Work.THWWorkStation.TCtrlWork.xWP_Analyse_StopAutomat:=FALSE;
		END_IF;
	END_CASE;
ELSE
	iSetTimeStamp_End:=1;
END_IF;
IF (diActual_NumberHoleToWork > 0) THEN
	FOR ii:=1 TO ciMaxWP DO
		IF (T_PartAnalysis.adiNumberHole[ii] = diActual_NumberHoleToWork) THEN
			diHoleNumber:=ii;
			EXIT;
		END_IF;
	END_FOR;
	IF (diHoleNumber = 0) OR (diHoleNumber > ciMaxWP) THEN
		diHoleNumber:=1;
	END_IF;
ELSE
	diHoleNumber:=1;
END_IF;
IF TStation_Work.THWWorkStation.TCtrlWork.xWP_Analyse_ActiveCycle AND NOT(gT_SafetyStatus.xSetupOperateModeActive) THEN
	TONCycleTime(IN:=TRUE,PT:=T#999999s);
	IF NOT(xInitCycleTime) THEN
		xInitCycleTime:=TRUE;
		tSaveCycleTime:=DINT_TO_TIME(T_PartAnalysis.adiCycleTime[diHoleNumber]);
	END_IF;
	T_PartAnalysis.adiCycleTime[diHoleNumber]:=TIME_TO_DINT(TONCycleTime.ET+tSaveCycleTime);
	IF (gxCentringActive OR gxOnlyCentringActive) AND NOT(TStation_Work.THWWorkStation.TCtrlWork.xWP_Analyse_ActiveWork) AND gxWP_Analyse_ActiveCentering THEN
		T_PartAnalysis.aiHCCounterCentering[diHoleNumber]:=iHCCounterCentering_Save + TStation_Work.THWWorkStation.TCtrlWork.iOverLimitCounterCentering;
	ELSE
		iHCCounterCentering_Save:=T_PartAnalysis.aiHCCounterCentering[diHoleNumber];
	END_IF;
ELSE
	TONCycleTime(IN:=FALSE);
	xInitCycleTime:=FALSE;
	tSaveCycleTime:=T#0s;
END_IF;

IF (TStation_Work.THWWorkStation.TCtrlWork.xWP_Analyse_ActiveWork AND NOT(gT_SafetyStatus.xSetupOperateModeActive)) OR gxSetPartQuality THEN
	IF NOT(gxSetPartQuality) THEN
		TONWorkTime(IN:=TRUE,PT:=T#999999s);
		IF NOT(xInitWorkTime) THEN
			xInitWorkTime:=TRUE;
			tSaveWorkTime:=DINT_TO_TIME(T_PartAnalysis.adiWorkTime[diHoleNumber]);
		END_IF;
	END_IF;
	IF NOT(gxSetPartQuality) THEN
		T_PartAnalysis.adiWorkTime[diHoleNumber]:=TIME_TO_DINT(TONWorkTime.ET+tSaveWorkTime);
	END_IF;
	T_PartAnalysis.abWorkPartQuality[diHoleNumber]:=TStation_Work.THWWorkStation.TCtrlWork.bPartQuality;
	IF TStation_Work.THWWorkStation.TCtrlWork.xWP_Analyse_ReadyToReadData THEN
		IF (T_PartAnalysis.arFirstHC[diHoleNumber] = 0.0) THEN
			T_PartAnalysis.arFirstHC[diHoleNumber]:=TStation_Work.THWWorkStation.TCtrlWork.rActualFirstContactPosition;
		END_IF;
		T_PartAnalysis.aiHCCounter[diHoleNumber]:=iHCCounter_Save + TStation_Work.THWWorkStation.TCtrlWork.iOverLimitCounter;
		T_PartAnalysis.aiHCCounterTorque[diHoleNumber]:=iHCCounterTorque_Save + TStation_Work.THWWorkStation.TCtrlWork.iOverLimitCounterTorque;
		T_PartAnalysis.aiHCCounterSpeed[diHoleNumber]:=iHCCounterSpeed_Save + TStation_Work.THWWorkStation.TCtrlWork.iOverLimitCounterSpeed;
	ELSE
		iHCCounter_Save:=T_PartAnalysis.aiHCCounter[diHoleNumber];
		iHCCounterTorque_Save:=T_PartAnalysis.aiHCCounterTorque[diHoleNumber];
		iHCCounterSpeed_Save:=T_PartAnalysis.aiHCCounterSpeed[diHoleNumber];
	END_IF;
	gxSetPartQuality:=FALSE;
	IF TStation_Work_St1.THWWorkStation.TCtrlWork.xWorkingFinished THEN
		TStation_Work.THWWorkStation.TCtrlWork.xWP_Analyse_ActiveWork:=FALSE;
	END_IF;
ELSE
	TONWorkTime(IN:=FALSE);
	xInitWorkTime:=FALSE;
	tSaveWorkTime:=T#0s;
	TStation_Work.THWWorkStation.TCtrlWork.xWP_Analyse_ReadyToReadData:=FALSE;
END_IF;

IF gxAddInfeedZ THEN
	IF (diHoleNumber <> 0) THEN
		IF gxAddInfeedZ THEN
			T_PartAnalysis.abInfeedCounterZ[diHoleNumber]:=T_PartAnalysis.abInfeedCounterZ[diHoleNumber] + 1;
		END_IF;
	END_IF;
	gxAddInfeedZ:=FALSE;
END_IF;

IF gxResetDataAnalysis_St1 THEN
	gxResetDataAnalysis_St1:=FALSE;
	T_PartAnalysis.sEndOfProcess:='';
	T_PartAnalysis.sStartOfProcess:='';
	T_PartAnalysis.diActual_NumberHoleToWork:=0;
	FOR ii:=1 TO ciMaxWP DO
		T_PartAnalysis.abWorkPartQuality[ii]:=0;
		T_PartAnalysis.adiCycleTime[ii]:=0;
		T_PartAnalysis.adiWorkTime[ii]:=0;
		T_PartAnalysis.aiHCCounter[ii]:=0;
		T_PartAnalysis.aiHCCounterCentering[ii]:=0;
		T_PartAnalysis.aiHCCounterTorque[ii]:=0;
		T_PartAnalysis.aiHCCounterSpeed[ii]:=0;
		T_PartAnalysis.arFirstHC[ii]:=0.0;
		T_PartAnalysis.abInfeedCounterZ[ii]:=0;
		T_PartAnalysis.adiNumberHole[ii]:=ii;
	END_FOR;
	T_PartAnalysis.sFileName:='';
END_IF;
IF (T_PartAnalysis.adiNumberHole[1] = 0) THEN
	FOR ii:=1 TO ciMaxWP DO
		T_PartAnalysis.adiNumberHole[ii]:=ii;
	END_FOR;
END_IF;
END_FUNCTION_BLOCK

(* POU PRG_LAYER4_PROCESS/FBPROCESS/FB_PreWarning_Ctrl_Message, ST *)
FUNCTION_BLOCK FB_PreWarning_Ctrl_Message
VAR_INPUT
	xPreWarninMessageBoxActive:BOOL;
END_VAR
VAR_IN_OUT
	T_PreWarning:ST_PREWARNING;
END_VAR
VAR_OUTPUT
END_VAR
VAR
	asMessageStringEngl:ARRAY [1..10,1..5] OF STRING(55);
	asMessageStringGer:ARRAY [1..10,1..5] OF STRING(55);
	FBPreWarningMessage: FB_PreWarning_Message;
	xInitMessageText: BOOL;
	RisingEdge_Message1: R_TRIG;
	RisingEdge_Message2: R_TRIG;
	FaillingEdge_Message1: F_TRIG;
	FaillingEdge_Message2: F_TRIG;
	ii: INT;
	iMessagePointer: INT;
	iNumberMessage: INT;
	aiSetMessageNumber:ARRAY [1..10] OF INT;
	asCopyMessageStringEngl:ARRAY [1..10,1..5] OF STRING(55);
	asCopyMessageStringGer:ARRAY [1..10,1..5] OF STRING(55);
	asDeleteMessageString:ARRAY [1..10,1..5] OF STRING(55);
	aiCopyMessageNrBuffer:ARRAY [1..10] OF INT;
	aiDeleteMessageNrBuffer:ARRAY [1..10] OF INT;
	jj: INT;
	xMessageExist: BOOL;
	iDeleteMessage: INT;
	iSaveDeleteMessage:ARRAY [1..12] OF INT;
	iSaveArrayNrMessage:INT:=0;
	FaillingEdgeDeleteWarningByMessageBox: F_TRIG;
	iSetMessageNumber: INT:=0;
	xForceDeleteMessage: BOOL;
END_VAR
IF NOT(xInitMessageText) THEN
	(* Initialisierung der Texte für die Vorwarnungen *)
	xInitMessageText:=TRUE;
	FBPreWarningMessage(	asMessageStringEngl:=asMessageStringEngl,
							asEmptyMessageEngl:=T_PreWarning.asEmptyMessageEngl,
							asMessageStringGer:=asMessageStringGer,
							asEmptyMessageGer:=T_PreWarning.asEmptyMessageGer);
END_IF;

IF (giDeleteMessageNumber <> 0) THEN
	iDeleteMessage:=0;
	FOR ii:=1 TO 10 DO
		IF (T_PreWarning.aiMessageNrBuffer[ii] = T_PreWarning.aiDeleteMessage[giDeleteMessageNumber]) THEN
			iSaveArrayNrMessage:=iSaveArrayNrMessage + 1;
			iSaveDeleteMessage[iSaveArrayNrMessage]:=T_PreWarning.aiDeleteMessage[giDeleteMessageNumber];
			iDeleteMessage:=ii;
			EXIT;
		END_IF;
	END_FOR;
	IF (iDeleteMessage <> 0) THEN
		T_PreWarning.asMessageBufferEngl[iDeleteMessage,1]:='';
		T_PreWarning.asMessageBufferEngl[iDeleteMessage,2]:='';
		T_PreWarning.asMessageBufferEngl[iDeleteMessage,3]:='';
		T_PreWarning.asMessageBufferEngl[iDeleteMessage,4]:='';
		T_PreWarning.asMessageBufferEngl[iDeleteMessage,5]:='';
		T_PreWarning.asMessageBufferGer[iDeleteMessage,1]:='';
		T_PreWarning.asMessageBufferGer[iDeleteMessage,2]:='';
		T_PreWarning.asMessageBufferGer[iDeleteMessage,3]:='';
		T_PreWarning.asMessageBufferGer[iDeleteMessage,4]:='';
		T_PreWarning.asMessageBufferGer[iDeleteMessage,5]:='';
		T_PreWarning.aiMessageNrBuffer[iDeleteMessage]:=0;
		asCopyMessageStringEngl:=asDeleteMessageString;
		asCopyMessageStringGer:=asDeleteMessageString;
		aiCopyMessageNrBuffer:=aiDeleteMessageNrBuffer;
		jj:=1;
		FOR ii:=1 TO 10 DO
			IF (T_PreWarning.asMessageBufferEngl[ii,1] <> '') THEN
				asCopyMessageStringEngl[jj,1]:=T_PreWarning.asMessageBufferEngl[ii,1];
				asCopyMessageStringEngl[jj,2]:=T_PreWarning.asMessageBufferEngl[ii,2];
				asCopyMessageStringEngl[jj,3]:=T_PreWarning.asMessageBufferEngl[ii,3];
				asCopyMessageStringEngl[jj,4]:=T_PreWarning.asMessageBufferEngl[ii,4];
				asCopyMessageStringEngl[jj,5]:=T_PreWarning.asMessageBufferEngl[ii,5];
				asCopyMessageStringGer[jj,1]:=T_PreWarning.asMessageBufferGer[ii,1];
				asCopyMessageStringGer[jj,2]:=T_PreWarning.asMessageBufferGer[ii,2];
				asCopyMessageStringGer[jj,3]:=T_PreWarning.asMessageBufferGer[ii,3];
				asCopyMessageStringGer[jj,4]:=T_PreWarning.asMessageBufferGer[ii,4];
				asCopyMessageStringGer[jj,5]:=T_PreWarning.asMessageBufferGer[ii,5];
				aiCopyMessageNrBuffer[jj]:=T_PreWarning.aiMessageNrBuffer[ii];
				jj:=jj + 1;
			END_IF;
		END_FOR;
		T_PreWarning.asMessageBufferEngl:=asCopyMessageStringEngl;
		T_PreWarning.asMessageBufferGer:=asCopyMessageStringGer;
		T_PreWarning.aiMessageNrBuffer:=aiCopyMessageNrBuffer;
	END_IF;
	 T_PreWarning.aiDeleteMessage[giDeleteMessageNumber]:=0;
	giDeleteMessageNumber:=giDeleteMessageNumber - 1;
	IF (giDeleteMessageNumber > 10) THEN
		giDeleteMessageNumber:=0;
	END_IF;
	IF NOT(xPreWarninMessageBoxActive) THEN
		xForceDeleteMessage:=TRUE;
	END_IF;
END_IF;

FaillingEdgeDeleteWarningByMessageBox(CLK:=xPreWarninMessageBoxActive);
IF FaillingEdgeDeleteWarningByMessageBox.Q OR xForceDeleteMessage THEN
	xForceDeleteMessage:=FALSE;
	FOR ii:=1 TO 10 DO
		IF (iSaveDeleteMessage[ii] =1) THEN
			T_PreWarning.xToolNearChangeSt1:=FALSE;
		ELSIF (iSaveDeleteMessage[ii] =2) THEN
			T_PreWarning.xZAxisBrakeBlockedSt1:=FALSE;
		END_IF;
		iSaveDeleteMessage[ii]:=0;
	END_FOR;;
	iSaveArrayNrMessage:=0;
END_IF;

(* aiSetMessageNumber:=0; *)
RisingEdge_Message1(CLK:=T_PreWarning.xToolNearChangeSt1);
IF RisingEdge_Message1.Q THEN
	iSetMessageNumber:=iSetMessageNumber + 1;
	aiSetMessageNumber[iSetMessageNumber]:=1;	(* Wz Wechsel für Station 1 muss bald vorgenommen werden! Beim erreichen max Anz. WzZyklen->Maschinen Stillstand! OK für Meldung Quittieren! RESET für ausgewählte Meldung Löschen! *)
END_IF;
RisingEdge_Message2(CLK:=T_PreWarning.xZAxisBrakeBlockedSt1);
IF RisingEdge_Message2.Q THEN
	iSetMessageNumber:=iSetMessageNumber + 1;
	aiSetMessageNumber[iSetMessageNumber]:=2;	(* Z Achsenbremse von Station 1 ist blockiert!' Lösen Sie Bitte die Handblockierung der Z Achse. OK für Meldung Quittieren! RESET für ausgewählte Meldung Löschen! *)
END_IF;

FaillingEdge_Message1(CLK:=T_PreWarning.xToolNearChangeSt1);
IF FaillingEdge_Message1.Q THEN
	giDeleteMessageNumber:=giDeleteMessageNumber + 1;
	T_PreWarning.aiDeleteMessage[giDeleteMessageNumber]:=2;	(* Löschen: Wz Wechsel für Station 1 muss bald vorgenommen werden! Beim erreichen max Anz. WzZyklen->Maschinen Stillstand! OK für Meldung Quittieren! RESET für ausgewählte Meldung Löschen! *)
END_IF;
FaillingEdge_Message2(CLK:=T_PreWarning.xZAxisBrakeBlockedSt1);
IF FaillingEdge_Message2.Q THEN
	TStation_Work_St1.THWWorkStation.TCtrlWork.xZAxisBrakeBlocked:=FALSE;
	giDeleteMessageNumber:=giDeleteMessageNumber + 1;
	T_PreWarning.aiDeleteMessage[giDeleteMessageNumber]:=6;	(* Löschen: Z Achsenbremse von Station 1 ist blockiert!' Lösen Sie Bitte die Handblockierung der Z Achse. OK für Meldung Quittieren! RESET für ausgewählte Meldung Löschen! *)
END_IF;

IF (T_NovRAM.T_Parameter.T_StationWork[gciStationSt1].T_ToolCounter.diMaxNumberToolCycle <> 0) AND
	(T_NovRAM.T_Parameter.T_StationWork[gciStationSt1].T_ToolCounter.diWarningAtToolCycleCounter <> 0) THEN
	IF (T_NovRAM.T_Parameter.T_StationWork[gciStationSt1].T_ToolCounter.diToolCycleCounter >= T_NovRAM.T_Parameter.T_StationWork[gciStationSt1].T_ToolCounter.diWarningAtToolCycleCounter) AND
	     (T_NovRAM.T_Parameter.T_StationWork[gciStationSt1].T_ToolCounter.diToolCycleCounter < T_NovRAM.T_Parameter.T_StationWork[gciStationSt1].T_ToolCounter.diMaxNumberToolCycle) THEN
		T_PreWarning.xToolNearChangeSt1:=TRUE;
	ELSE
		T_PreWarning.xToolNearChangeSt1:=FALSE;
	END_IF;
ELSE
	T_PreWarning.xToolNearChangeSt1:=FALSE;		(* WzZähler ist ausgeschaltet und darf daher auch keine Meldung ausgeben *)
END_IF;
IF TStation_Work_St1.THWWorkStation.TCtrlWork.xZAxisBrakeBlocked THEN
	T_PreWarning.xZAxisBrakeBlockedSt1:=TRUE;
ELSE
	T_PreWarning.xZAxisBrakeBlockedSt1:=FALSE;
END_IF;

iMessagePointer:=1;	(* Dies besagt die Stelle wo eine Meldung eingetragen werden *)
iNumberMessage:=0;	(* Dies besagt wieviele Meldungen im Buffer vorhanden sind *)
(* Überprüfe wieviele Meldungen im Buffer abgelegt sind *)
FOR ii:=1 TO 10 DO
	IF T_PreWarning.asMessageBufferEngl[ii,1] <> '' THEN
		iNumberMessage:=iNumberMessage + 1;
		IF (iMessagePointer < 10) THEN
			iMessagePointer:=iMessagePointer + 1;
		END_IF;
	END_IF;
END_FOR;
IF (iNumberMessage <> 0) THEN T_PreWarning.xPreWarningActive:=TRUE; ELSE T_PreWarning.xPreWarningActive:=FALSE; END_IF;
T_PreWarning.iNumberOfMessage:=iNumberMessage;
IF (iSetMessageNumber <> 0) THEN
	xMessageExist:=FALSE;
	(* Überprüfe zuerst ob es nicht schon die gleiche Meldung gibt *)
	FOR ii:=1 TO 10 DO
		IF (T_PreWarning.aiMessageNrBuffer[ii] = aiSetMessageNumber[iSetMessageNumber]) THEN
			xMessageExist:=TRUE;
			EXIT;
		END_IF;
	END_FOR;
	IF NOT(xMessageExist) THEN
		T_PreWarning.asMessageBufferEngl[iMessagePointer,1]:=asMessageStringEngl[aiSetMessageNumber[iSetMessageNumber],1];
		T_PreWarning.asMessageBufferEngl[iMessagePointer,2]:=asMessageStringEngl[aiSetMessageNumber[iSetMessageNumber],2];
		T_PreWarning.asMessageBufferEngl[iMessagePointer,3]:=asMessageStringEngl[aiSetMessageNumber[iSetMessageNumber],3];
		T_PreWarning.asMessageBufferEngl[iMessagePointer,4]:=asMessageStringEngl[aiSetMessageNumber[iSetMessageNumber],4];
		T_PreWarning.asMessageBufferEngl[iMessagePointer,5]:=asMessageStringEngl[aiSetMessageNumber[iSetMessageNumber],5];
		T_PreWarning.asMessageBufferGer[iMessagePointer,1]:=asMessageStringGer[aiSetMessageNumber[iSetMessageNumber],1];
		T_PreWarning.asMessageBufferGer[iMessagePointer,2]:=asMessageStringGer[aiSetMessageNumber[iSetMessageNumber],2];
		T_PreWarning.asMessageBufferGer[iMessagePointer,3]:=asMessageStringGer[aiSetMessageNumber[iSetMessageNumber],3];
		T_PreWarning.asMessageBufferGer[iMessagePointer,4]:=asMessageStringGer[aiSetMessageNumber[iSetMessageNumber],4];
		T_PreWarning.asMessageBufferGer[iMessagePointer,5]:=asMessageStringGer[aiSetMessageNumber[iSetMessageNumber],5];
		T_PreWarning.aiMessageNrBuffer[iMessagePointer]:=aiSetMessageNumber[iSetMessageNumber];
	END_IF;
	aiSetMessageNumber[iSetMessageNumber]:=0;
	iSetMessageNumber:=iSetMessageNumber - 1;
	IF (iSetMessageNumber > 10) THEN
		iSetMessageNumber:=0;
	END_IF;
END_IF;
END_FUNCTION_BLOCK

(* POU PRG_LAYER4_PROCESS/FBPROCESS/FB_PreWarning_Message, ST *)
FUNCTION_BLOCK FB_PreWarning_Message
VAR_INPUT
END_VAR
VAR_IN_OUT
	asMessageStringEngl:ARRAY [1..10,1..5] OF STRING(55);
	asEmptyMessageEngl:ARRAY [1..5] OF STRING(55);
	asMessageStringGer:ARRAY [1..10,1..5] OF STRING(55);
	asEmptyMessageGer:ARRAY [1..5] OF STRING(55);
END_VAR
VAR_OUTPUT
END_VAR
VAR
	iMessageNr: INT;
END_VAR
(* ENGLISCH *)
asEmptyMessageEngl[1]:='Message 0 of 0';	(* Dieser Text wird Dynamisch erstellt und besagt welche Message von wievielen Messages ausgewählt wurde *)
asEmptyMessageEngl[2]:='No Pre Warning Message';
asEmptyMessageEngl[3]:='';
asEmptyMessageEngl[4]:='OK for acknowledge Message!';
asEmptyMessageEngl[5]:='RESET no effect!';
iMessageNr:=1;
asMessageStringEngl[iMessageNr,1]:='Message 1 of 1';	(* Dieser Text wird Dynamisch erstellt und besagt welche Message von wievielen Messages ausgewählt wurde *)
asMessageStringEngl[iMessageNr,2]:='Tool Change for Station 1 must be nearly occur!';
asMessageStringEngl[iMessageNr,3]:='On reach of max. Number ToolCycle->Automat stop!';
asMessageStringEngl[iMessageNr,4]:='OK for acknowledge Message!';
asMessageStringEngl[iMessageNr,5]:='RESET for delete selected Message!';
iMessageNr:=iMessageNr + 1;
asMessageStringEngl[iMessageNr,1]:='Message 2 of 2';	(* Dieser Text wird Dynamisch erstellt und besagt welche Message von wievielen Messages ausgewählt wurde *)
asMessageStringEngl[iMessageNr,2]:='Z Axis brake of Station 1 is blocked!';
asMessageStringEngl[iMessageNr,3]:='Please release the Manual block of the Z Axis.';
asMessageStringEngl[iMessageNr,4]:='OK for acknowledge Message!';
asMessageStringEngl[iMessageNr,5]:='RESET for delete selected Message!';
iMessageNr:=iMessageNr + 1;
asMessageStringEngl[iMessageNr,1]:='Message 3 of 3';	(* Dieser Text wird Dynamisch erstellt und besagt welche Message von wievielen Messages ausgewählt wurde *)
asMessageStringEngl[iMessageNr,2]:='';
asMessageStringEngl[iMessageNr,3]:='';
asMessageStringEngl[iMessageNr,4]:='OK for acknowledge Message!';
asMessageStringEngl[iMessageNr,5]:='RESET for delete selected Message!';
iMessageNr:=iMessageNr + 1;
asMessageStringEngl[iMessageNr,1]:='Message 4 of 4';	(* Dieser Text wird Dynamisch erstellt und besagt welche Message von wievielen Messages ausgewählt wurde *)
asMessageStringEngl[iMessageNr,2]:='';
asMessageStringEngl[iMessageNr,3]:='';
asMessageStringEngl[iMessageNr,4]:='OK for acknowledge Message!';
asMessageStringEngl[iMessageNr,5]:='RESET for delete selected Message!';
iMessageNr:=iMessageNr + 1;
asMessageStringEngl[iMessageNr,1]:='Message 5 of 5';	(* Dieser Text wird Dynamisch erstellt und besagt welche Message von wievielen Messages ausgewählt wurde *)
asMessageStringEngl[iMessageNr,2]:='';
asMessageStringEngl[iMessageNr,3]:='';
asMessageStringEngl[iMessageNr,4]:='OK for acknowledge Message!';
asMessageStringEngl[iMessageNr,5]:='RESET for delete selected Message!';
iMessageNr:=iMessageNr + 1;
asMessageStringEngl[iMessageNr,1]:='Message 6 of 6';	(* Dieser Text wird Dynamisch erstellt und besagt welche Message von wievielen Messages ausgewählt wurde *)
asMessageStringEngl[iMessageNr,2]:='';
asMessageStringEngl[iMessageNr,3]:='';
asMessageStringEngl[iMessageNr,4]:='OK for acknowledge Message!';
asMessageStringEngl[iMessageNr,5]:='RESET for delete selected Message!';
iMessageNr:=iMessageNr + 1;
asMessageStringEngl[iMessageNr,1]:='Message 7 of 7';	(* Dieser Text wird Dynamisch erstellt und besagt welche Message von wievielen Messages ausgewählt wurde *)
asMessageStringEngl[iMessageNr,2]:='';
asMessageStringEngl[iMessageNr,3]:='';
asMessageStringEngl[iMessageNr,4]:='OK for acknowledge Message!';
asMessageStringEngl[iMessageNr,5]:='RESET for delete selected Message!';
iMessageNr:=iMessageNr + 1;
asMessageStringEngl[iMessageNr,1]:='Message 8 of 8';	(* Dieser Text wird Dynamisch erstellt und besagt welche Message von wievielen Messages ausgewählt wurde *)
asMessageStringEngl[iMessageNr,2]:='';
asMessageStringEngl[iMessageNr,3]:='';
asMessageStringEngl[iMessageNr,4]:='OK for acknowledge Message!';
asMessageStringEngl[iMessageNr,5]:='RESET for delete selected Message!';
iMessageNr:=iMessageNr + 1;
asMessageStringEngl[iMessageNr,1]:='Message 9 of 9';	(* Dieser Text wird Dynamisch erstellt und besagt welche Message von wievielen Messages ausgewählt wurde *)
asMessageStringEngl[iMessageNr,2]:='';
asMessageStringEngl[iMessageNr,3]:='';
asMessageStringEngl[iMessageNr,4]:='OK for acknowledge Message!';
asMessageStringEngl[iMessageNr,5]:='RESET for delete selected Message!';
iMessageNr:=iMessageNr + 1;
asMessageStringEngl[iMessageNr,1]:='Message 10 of 10';	(* Dieser Text wird Dynamisch erstellt und besagt welche Message von wievielen Messages ausgewählt wurde *)
asMessageStringEngl[iMessageNr,2]:='';
asMessageStringEngl[iMessageNr,3]:='';
asMessageStringEngl[iMessageNr,4]:='OK for acknowledge Message!';
asMessageStringEngl[iMessageNr,5]:='RESET for delete selected Message!';

(* DEUTSCH *)
asEmptyMessageGer[1]:='Meldung 0 von 0';	(* Dieser Text wird Dynamisch erstellt und besagt welche Message von wievielen Messages ausgewählt wurde *)
asEmptyMessageGer[2]:='Es bestehen keine Warnungen';
asEmptyMessageGer[3]:='';
asEmptyMessageGer[4]:='OK für Meldung Quittieren!';
asEmptyMessageGer[5]:='RESET hat keine Auswirkung!';
iMessageNr:=1;
asMessageStringGer[iMessageNr,1]:='Meldung 1 von 1';	(* Dieser Text wird Dynamisch erstellt und besagt welche Message von wievielen Messages ausgewählt wurde *)
asMessageStringGer[iMessageNr,2]:='Wz Wechsel für Station 1 muss bald vorgenommen werden!';
asMessageStringGer[iMessageNr,3]:='Beim erreichen max Anz. WzZyklen->Maschinen Stillstand!';
asMessageStringGer[iMessageNr,4]:='OK für Meldung Quittieren!';
asMessageStringGer[iMessageNr,5]:='RESET für ausgewählte Meldung Löschen!';
iMessageNr:=iMessageNr + 1;
asMessageStringGer[iMessageNr,1]:='Meldung 2 von 2';	(* Dieser Text wird Dynamisch erstellt und besagt welche Message von wievielen Messages ausgewählt wurde *)
asMessageStringGer[iMessageNr,2]:='Z Achsenbremse von Station 1 ist blockiert!';
asMessageStringGer[iMessageNr,3]:='Lösen Sie Bitte die Handblockierung der Z Achse.';
asMessageStringGer[iMessageNr,4]:='OK für Meldung Quittieren!';
asMessageStringGer[iMessageNr,5]:='RESET für ausgewählte Meldung Löschen!';
iMessageNr:=iMessageNr + 1;
asMessageStringGer[iMessageNr,1]:='Meldung 3 von 3';	(* Dieser Text wird Dynamisch erstellt und besagt welche Message von wievielen Messages ausgewählt wurde *)
asMessageStringGer[iMessageNr,2]:='';
asMessageStringGer[iMessageNr,3]:='';
asMessageStringGer[iMessageNr,4]:='OK für Meldung Quittieren!';
asMessageStringGer[iMessageNr,5]:='RESET für ausgewählte Meldung Löschen!';
iMessageNr:=iMessageNr + 1;
asMessageStringGer[iMessageNr,1]:='Meldung 4 von 4';	(* Dieser Text wird Dynamisch erstellt und besagt welche Message von wievielen Messages ausgewählt wurde *)
asMessageStringGer[iMessageNr,2]:='';
asMessageStringGer[iMessageNr,3]:='';
asMessageStringGer[iMessageNr,4]:='OK für Meldung Quittieren!';
asMessageStringGer[iMessageNr,5]:='RESET für ausgewählte Meldung Löschen!';
iMessageNr:=iMessageNr + 1;
asMessageStringGer[iMessageNr,1]:='Meldung 5 von 5';	(* Dieser Text wird Dynamisch erstellt und besagt welche Message von wievielen Messages ausgewählt wurde *)
asMessageStringGer[iMessageNr,2]:='';
asMessageStringGer[iMessageNr,3]:='';
asMessageStringGer[iMessageNr,4]:='OK für Meldung Quittieren!';
asMessageStringGer[iMessageNr,5]:='RESET für ausgewählte Meldung Löschen!';
iMessageNr:=iMessageNr + 1;
asMessageStringGer[iMessageNr,1]:='Meldung 6 von 6';	(* Dieser Text wird Dynamisch erstellt und besagt welche Message von wievielen Messages ausgewählt wurde *)
asMessageStringGer[iMessageNr,2]:='';
asMessageStringGer[iMessageNr,3]:='';
asMessageStringGer[iMessageNr,4]:='OK für Meldung Quittieren!';
asMessageStringGer[iMessageNr,5]:='RESET für ausgewählte Meldung Löschen!';
iMessageNr:=iMessageNr + 1;
asMessageStringGer[iMessageNr,1]:='Meldung 7 von 7';	(* Dieser Text wird Dynamisch erstellt und besagt welche Message von wievielen Messages ausgewählt wurde *)
asMessageStringGer[iMessageNr,2]:='';
asMessageStringGer[iMessageNr,3]:='';
asMessageStringGer[iMessageNr,4]:='OK für Meldung Quittieren!';
asMessageStringGer[iMessageNr,5]:='RESET für ausgewählte Meldung Löschen!';
iMessageNr:=iMessageNr + 1;
asMessageStringGer[iMessageNr,1]:='Meldung 8 von 8';	(* Dieser Text wird Dynamisch erstellt und besagt welche Message von wievielen Messages ausgewählt wurde *)
asMessageStringGer[iMessageNr,2]:='';
asMessageStringGer[iMessageNr,3]:='';
asMessageStringGer[iMessageNr,4]:='OK für Meldung Quittieren!';
asMessageStringGer[iMessageNr,5]:='RESET für ausgewählte Meldung Löschen!';
iMessageNr:=iMessageNr + 1;
asMessageStringGer[iMessageNr,1]:='Meldung 9 von 9';	(* Dieser Text wird Dynamisch erstellt und besagt welche Message von wievielen Messages ausgewählt wurde *)
asMessageStringGer[iMessageNr,2]:='';
asMessageStringGer[iMessageNr,3]:='';
asMessageStringGer[iMessageNr,4]:='OK für Meldung Quittieren!';
asMessageStringGer[iMessageNr,5]:='RESET für ausgewählte Meldung Löschen!';
iMessageNr:=iMessageNr + 1;
asMessageStringGer[iMessageNr,1]:='Meldung 10 von 10';	(* Dieser Text wird Dynamisch erstellt und besagt welche Message von wievielen Messages ausgewählt wurde *)
asMessageStringGer[iMessageNr,2]:='';
asMessageStringGer[iMessageNr,3]:='';
asMessageStringGer[iMessageNr,4]:='OK für Meldung Quittieren!';
asMessageStringGer[iMessageNr,5]:='RESET für ausgewählte Meldung Löschen!';
END_FUNCTION_BLOCK

(* POU PRG_LAYER3_STATION/PRG_STATION_WORK_ST1, FBD *)
PROGRAM PRG_STATION_WORK_ST1
VAR
	FBStationWork_St1: FB_STATION_WORK;
	xActive_Work_St1: BOOL;
	xRdy_Work_St1: BOOL;
	xEnd_Work_St1: BOOL;
	xStop_Work_St1: BOOL;
	xReferenced_Work_St1: BOOL;
	xError_Work_St1: BOOL;
	iErrorNr_Work_St1: DINT;
	iStatusFctNr_Work_St1 : INT;
	xStationPowerON_St1: BOOL;
	xAxisBrakeBlock_St1:BOOL;
END_VAR
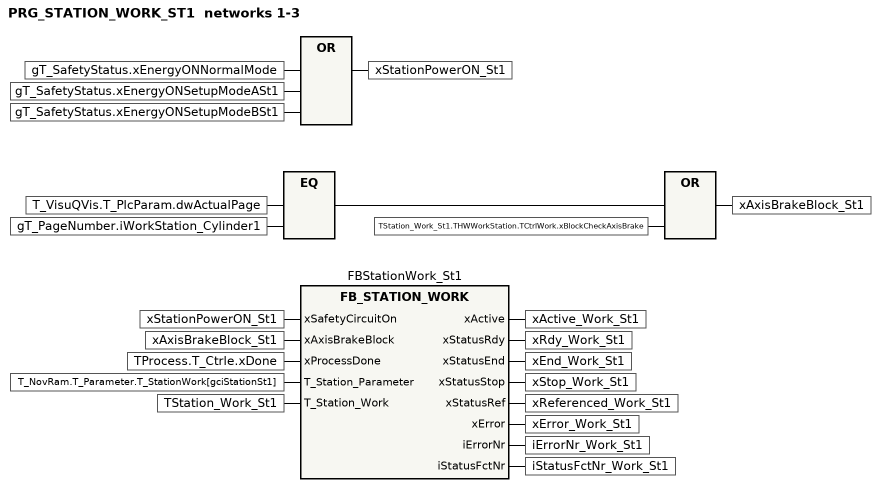
_FBD_ (* Function Block Diagram *)
NETWORK 1
	OR(gT_SafetyStatus.xEnergyONNormalMode, gT_SafetyStatus.xEnergyONSetupModeASt1, gT_SafetyStatus.xEnergyONSetupModeBSt1) => xStationPowerON_St1
NETWORK 2
	OR(EQ(T_VisuQVis.T_PlcParam.dwActualPage, gT_PageNumber.iWorkStation_Cylinder1), TStation_Work_St1.THWWorkStation.TCtrlWork.xBlockCheckAxisBrake) => xAxisBrakeBlock_St1
NETWORK 3
	FBStationWork_St1:FB_STATION_WORK(xSafetyCircuitOn: xStationPowerON_St1, xAxisBrakeBlock: xAxisBrakeBlock_St1, xProcessDone: TProcess.T_Ctrle.xDone, T_Station_Parameter: T_NovRam.T_Parameter.T_StationWork[gciStationSt1], T_Station_Work: TStation_Work_St1, xStatusRdy => xRdy_Work_St1, xStatusEnd => xEnd_Work_St1, xStatusStop => xStop_Work_St1, xStatusRef => xReferenced_Work_St1, xError => xError_Work_St1, iErrorNr => iErrorNr_Work_St1, iStatusFctNr => iStatusFctNr_Work_St1) => xActive_Work_St1
_END_FBD_
(* the same logic as Structured Text *)
(* Network 1 *)
xStationPowerON_St1 := gT_SafetyStatus.xEnergyONNormalMode OR gT_SafetyStatus.xEnergyONSetupModeASt1 OR gT_SafetyStatus.xEnergyONSetupModeBSt1;
(* Network 2 *)
xAxisBrakeBlock_St1 := (T_VisuQVis.T_PlcParam.dwActualPage = gT_PageNumber.iWorkStation_Cylinder1) OR TStation_Work_St1.THWWorkStation.TCtrlWork.xBlockCheckAxisBrake;
(* Network 3 *)
FBStationWork_St1(xSafetyCircuitOn := xStationPowerON_St1, xAxisBrakeBlock := xAxisBrakeBlock_St1, xProcessDone := TProcess.T_Ctrle.xDone, T_Station_Parameter := T_NovRam.T_Parameter.T_StationWork[gciStationSt1], T_Station_Work := TStation_Work_St1);
xRdy_Work_St1 := FBStationWork_St1.xStatusRdy;
xEnd_Work_St1 := FBStationWork_St1.xStatusEnd;
xStop_Work_St1 := FBStationWork_St1.xStatusStop;
xReferenced_Work_St1 := FBStationWork_St1.xStatusRef;
xError_Work_St1 := FBStationWork_St1.xError;
iErrorNr_Work_St1 := FBStationWork_St1.iErrorNr;
iStatusFctNr_Work_St1 := FBStationWork_St1.iStatusFctNr;
xActive_Work_St1 := FBStationWork_St1.xActive;
END_PROGRAM

(* POU PRG_LAYER3_STATION/FBSTATIONEN/FB_STATION_WORK, ST *)
FUNCTION_BLOCK FB_STATION_WORK
VAR_INPUT
	xSafetyCircuitOn:BOOL;
	xAxisBrakeBlock:BOOL;		(* Blockieren der automatischen überwachung der Achsenbremsen *)
	xProcessDone:BOOL;
END_VAR
VAR_IN_OUT
	T_Station_Parameter: ST_RETAIN_DATA_STATIONWORK;
	T_Station_Work : ST_STATION;
END_VAR
VAR_OUTPUT
	xActive : BOOL :=FALSE;
	xStatusRdy : BOOL := FALSE;
	xStatusEnd : BOOL := FALSE;
	xStatusStop : BOOL := FALSE;
	xStatusRef : BOOL := FALSE;
	xError : BOOL := FALSE;
	iErrorNr : DINT :=0;
	iStatusFctNr : INT := 0;
END_VAR
VAR
(* Pointer auf Actuatoren *)
	ptrTAxisZ 							:POINTER TO ST_AXIS;		(* Achse für die Hubachse *)
	ptrTAxisS 							:POINTER TO ST_AXIS;		(* Achse für die Werkzeugspindel *)
	ptrTCylToolDeflection					:POINTER TO ST_CYLINDER;	(* Servoventil für das bestimmen der vertikalen Auslenkraft *)
	ptrTCylToolTorqueHC 					:POINTER TO ST_CYLINDER;	(* Drehmomentueberwachung HC *)
	ptrTCylToolTorqueOverload 			:POINTER TO ST_CYLINDER;	(* Drehmomentueberwachung Ueberlast *)
	ptrTTorqueSensorMeasRange			:POINTER TO ST_CYLINDER;	(* Controlling fuer den Drehmomentsensor, Einstellung des Drehmomentbereiches *)	(* IGS *)
	ptrTTorqueSensorControl				:POINTER TO ST_CYLINDER;	(* Controlling fuer den Drehmomentsensor, Ueberprüfung auf Funktionalitaet *)			(* IGS *)
	ptrTSensorTorque 					:POINTER TO ST_CYLINDER;	(* Analoger Sensor für Drehmoment detektion *)								(* IGS *)
	ptrTSensorTorqueOverload 			:POINTER TO ST_CYLINDER;	(* Digitaler Sensor für Drehmoment Ueberlast detektion *)							(* IGS *)
	ptrTCylBrakeReleaseZAxis 				:POINTER TO ST_CYLINDER;	(* Zylinder für lösen der Bremse bei der Z Achse *)
	ptrTCylWorkpieceClamp				:POINTER TO ST_CYLINDER;	(* Ventil fuer Werkstueckfixierzylinder *)
	ptrTValveAirTable						:POINTER TO ST_CYLINDER;	(* Ventil fuer die Luft des Tisches *)
	ptrTValveVacuumTable				:POINTER TO ST_CYLINDER;	(* Ventil fuer Vacuum des Tisches *)
	ptrTValveCleanNozzle					:POINTER TO ST_CYLINDER;	(* Ventil fuer die Reinigungsduese*)											(* BEF *)
	ptrTAxisBubbler						:POINTER TO ST_DC_AXIS;	(* Ruehrwerk fuer Suspension *)												(* IGS3 *)
	ptrTAxisFeedPump					:POINTER TO ST_DC_AXIS;	(* Foerderpumpe fuer Suspension *)											(* IGS3 *)

	TDeleteStationStruct : ST_STATION;
	xTmpStopFunction: BOOL := FALSE;
	iStationFunctionNr: INT := 0;
(* Trigger *)
	fbFTrig: F_TRIG;
	fbRTrig: R_TRIG;
	xInitDelEnable: BOOL := FALSE;
	xReadyChkError: BOOL;
	xDontDeleteErrorFlag: BOOL;
	xInitStep: BOOL := FALSE;
	xInitSetEnable: BOOL := FALSE;
	xRdyDisableStation: BOOL;
	iStepEnable: INT := 0;
	xStartFunction: BOOL := FALSE;
	iMaxFunctionNr:INT:=10;
	xTmp: BOOL;
	xSetEnd: BOOL := FALSE;
	xSetError: BOOL;
	diErrorNumber: DINT;
	iCountCycle: INT;
	TONCheckAxisVoltagBooting: TON;
	xStartTimer: BOOL;
	xWaitAxisVoltageBooting: BOOL;
	TONWaitAxisCurrentSwitchON: TON;
	xSecurityCircuitOn: BOOL;
	xSecurityCircuitOff: BOOL;
	iStepSecCircuit: INT;
	xInitSecCircuit: BOOL;
	TONCheckError: TON;
	xStationError: BOOL := FALSE;
	xForceHWError: BOOL;
	xForceResetAxis: BOOL;
	xInitError: BOOL := FALSE;
	iSettledErrFromFunction: INT;
	xTmpStationError: BOOL;
	xAxisErrorActive: BOOL;
	TONWaitReset: TON;
	xStepError: BOOL;
	xReadyToQuitErr: BOOL;
	xTmpStart: BOOL := FALSE;
	xInitStart: BOOL := FALSE;
	xInitStop: BOOL := FALSE;
	xCheckAxisCurrent: BOOL;
	xStFct_Reset: BOOL;
	xStFct_SetEnd: BOOL;
	xStFct_End: BOOL;
	xStFct_Stop: BOOL;
	xStFct_Start: BOOL;
	xStFct_StartMainPrc: BOOL;
	iStFct_StepError: INT;
	xStFct_InitError: BOOL;
	xStFct_HardwareError: BOOL;
	diStFct_ErrorNr: DINT;
	diStFct_TmpErrorNr: DINT;
	xStFct_Error: BOOL;
	xStFct_QuitErr: BOOL;
	xStFct_Abord: BOOL;
	xStFct_ErrorActuator: BOOL;
	xStFct_ExecuteActuator: BOOL;
	xStFct_StartMainCtr: BOOL;
	xStFct_InitMainCtr: BOOL;
	iStFct_StepPrc: INT;
	xStFct_InitStep: BOOL;
	wStFct_Status: WORD;
	xStFct_TmpStop: BOOL;
	iStFct_TmpStopStep: INT;
	xStFct_Freeze: BOOL;
	xStFct_StartPrc_Parallel: BOOL;
	iStFct_StepPrc_Parallel: INT;
	xStFct_InitStep_Parallel: BOOL;
	xStFct_StopSlide: BOOL;
	fbStFct_CalcCuttingSpeed:FB_CalcCuttingSpeed;
	fbStFct_SparkOutProcess:FB_SparkOutProcess;
	xStFct_CapturePosition: BOOL;
	xStFct_ResetCalcCutSpeed: BOOL;
	xStFct_TmpActiveFirstHC: BOOL;
	xStFct_StartProcessTimer: BOOL;
	fbStFct_TONProcessMinTime: TON;
	xStFct_MinTimeProcessReady: BOOL;
	fbStFct_TONProcessMaxTime: TON;
	xStFct_TmpStopProcess: BOOL;
	xStFct_InitStopProcess: BOOL;
	iStFct_StopProcess: INT;
	xStFct_StartSparkOutProcess: BOOL;
	xStFct_ResetSparkOutProcess: BOOL;
	rStFct_TmpDiffOverLimitPosition: REAL;
	rStFct_StopPosition: REAL;
	iStFct_TmpHCStartPosCounter: INT;
	iStFct_TmpNumberTryInfeed: INT;
	rStFct_ForceDeflection: REAL;
	rStFct_ForceTorque: REAL;
	TONTimeOutEnablePart: TON;
	xStFct_PositionOutRange_Z: BOOL;
	iStFct_PosErrorNr: INT;
	xStFct_DeflCalibError: BOOL;
	xStFct_TorqueCalibError: BOOL;
	xStFct_ForceStationError: BOOL;
	iStFct_StepCollision: INT;
	xFirstBooting: BOOL;
	TONStFct_WaitAxisReady: TON;
	lrStFct_SaveAxisPosition: LREAL;
	xStFct_ForceSetSpeedZAxis: BOOL;
	xStFct_ForceSetSpeedTorqueZAxis: BOOL;
	xStFct_BlockWorking2: BOOL;
	xStFct_InitialCalcProcWork: BOOL;
	rStFct_ZSavePosition: REAL;
	rStFct_ZCalcDistance: REAL;
	diStFct_Counter: DINT;
	rStFct_CalcWorkForce: REAL;
	iStFct_StepMaxProcWork: INT;
	xStFct_ForceHC: BOOL;
	iStFct_StepZWorkSpeedRegulator: INT;
	rStFct_AddWorkForce: REAL;
	rStFct_CheckZSavePosition: REAL;
	iStFct_StepCheckToolBlock: INT;
	xStFct_HCActivated: BOOL;
	iStFct_StepCheckTorque: INT;
	iStFct_DataInputNr: INT;
	xStFct_ToolDeflectionActiveStopProcess: BOOL;
	xStFct_ToolClampInactiveStopProcess: BOOL;
	iStFct_StepWPRotate: INT;
	xStFct_WPRotated: BOOL;
	xStFct_ForceRotate: BOOL;
	iStFct_NumberWPRotate: INT;
	xStFct_Overload_StopProcess: BOOL;
	iStFct_Overload_StopProcess: INT;
	TONWorkTime: TON;
	iStFct_StepStartToolSpindle: INT;
	xStFct_InitStepStartToolSpindle: BOOL;
	iStFct_StepStopToolSpindle: INT;
	xStFct_InitStepStopToolSpindle: BOOL;
	rStFct_TmpOffsetDeflection: REAL;
	rStFct_TmpOffsetTorque: REAL;
	xStFct_TmpSaveOffset: BOOL;
	xStFct_SetForceToolDeflection: BOOL;
	iStFct_StepSetForceToolDeflection: INT;
	TONStFct_DeflectionSensorON: TON;
	TONStFct_DeflectionSensorOFF: TON;
	xStFct_DeflectionSensorON: BOOL;
	iStFct_ii: INT;
	xStFct_FirstTime: BOOL;
	tStFct_MaxTimeActiveFunction: TIME;
	fbStFct_TONChkMaxTimeActive: TON;
	fbStFct_TONWaitCycle: TON;
	tStFct_TimeSpindleActive: TIME;
	tStFct_TimeSpindleInactive: TIME;
	xSetSlowToFastSpeed: BOOL;
	rStFct_SetZHCPosition:REAL;
	xStFct_ToolDeflectionActiv: BOOL;
	xStFct_InitAxialSensor: BOOL;
	xStFct_CheckAxialSensor: BOOL;
	lrStFct_ActualPosition: LREAL;
	xStFct_ZAxisBrakeBlocked: BOOL;
	xMaxTorqueActive: BOOL;
	xPartDiscNotInPosition: BOOL;
	TONWaitCheckCylinder: TON;
	TONStFct_TorqueSensorOFF: TON;
	TONStFct_TorqueSensorON: TON;
	xStFct_TorqueSensorON: BOOL;
	xStFct_ToolTorqueCheckedOK: BOOL;
	xStFct_CheckState1: BOOL;
	xStFct_CheckState2: BOOL;
	xStFct_CheckActive1: BOOL;
	xStFct_CheckActive2: BOOL;
	xStFct_FirstTimeTorque: BOOL;
	xStFct_SetForceToolTorque: BOOL;
	iStFct_StepSetForceToolTorque: INT;
	xBlockCheckLimitSwitch: BOOL;
	TONCalcMinTimeEnable: TON;

	rTorquePercent: REAL;							(* IGS *)

	TONWaitReady:TON;							(* IGS *)
	rStFct_V1:REAL;								(* IGS *)
	rStFct_V2:REAL;								(* IGS *)
	rStFct_S1:REAL;								(* IGS *)
	rStFct_S2:REAL;								(* IGS *)
	rStFct_M:REAL;								(* IGS *)
	rTorqueForce:REAL;							(* IGS *)
	rActTorque:REAL;								(* IGS *)
	rTorqueMax:REAL;							(* IGS *)
	rTorqueMax_Max:REAL;						(* IGS *)
	rTorqueMin:REAL;								(* IGS *)
	rTorqueMin_Min:REAL;							(* IGS *)
	rStFct_CalcZSpeed:REAL;						(* IGS *)

	(* Progressive Stroke *)
	xStFct_ProgressStrokeReady:BOOL;				(* BEF *)
	xStFct_ProgressStrokeRunning:BOOL;			(* BEF *)
	iStFct_StepProgressStroke:INT;					(* BEF *)
	rStFct_ProgressStrokePosition:REAL;			(* BEF *)

	(* Spark Out *)
	xStFct_InitStepSparkOut:BOOL;					(* BEF *)
	xStFct_SparkOutRunning:BOOL;					(* BEF *)
	iStFct_StepSparkOut:INT;						(* BEF *)
	xStFct_ActiveChgForceDeflection:BOOL;			(* BEF *)
	xStFct_SetForceDeflection:BOOL;				(* BEF *)
	xStFct_InitSetForceDeflection:BOOL;				(* BEF *)
	iStFct_TmpCountHub:INT;						(* BEF *)
	xStFct_BlockCounter:BOOL;						(* BEF *)
	xStFct_RepeatProcess:BOOL;					(* BEF *)
	xStFct_InitSparkOutVar:BOOL;					(* BEF *)

	xStFct_SparkOutDone:BOOL;					(* BEF *)

	(* Controllers *)
	rStFct_CtrlInputWorkingSpeed:REAL;				(* BEF *) (* General speed, can be positive or negative *)

	(* Outfeed Stroke *)
	xStFct_OutfeedStrokeRunning:BOOL; 				(* BEF *)

	(* .HW_Axis_DC *)
(*	iStepBubbler:INT;															(* IGS3 *)
	iStepFeeder:INT;															(* IGS3 *)*)

	(* .StationFunction_Fct_07_Calibration2 *)
	TONStFct_WaitMeasure:TON;					(* IGS *)
	iStFct_MeasuringStep:INT;						(* IGS *)
	arStFct_NullPointToolTorque:ARRAY [1..20] OF REAL;	(* Durchschnittswert von 20 Messwerten wird der Nullpunkt bestimmt *)		(* IGS *)
	rStFct_NullPointToolTorque: REAL;				(* IGS *)
	TONWaitHCActive: TON;
	TONWaitHCInactive: TON;
	lrActualPositionSave: LREAL;
	lrZ1HCMinPosition: LREAL;
	lrZ1HCMaxPosition: LREAL;
	diHCCheckCounter: DINT;
	lrActualPositionSaveSwitchZSpeed: LREAL;
	TONWaitStopOAxis: TON;
	xZFastSpeedSettled: BOOL;

	TONCalcTorque: TON;
	diStepCount: DINT;
	rTorqueSpindleSensorSave: REAL;
	rTorqueSpindleSensor: REAL;
	rOutMaxLimit: REAL;
	rOutMinLimit: REAL;
	T_CtrlPara: ST_CTRL_PID_PARAM;
	FBPIDCTRL: FB_PID_CONTROL;
	T_CtrlPara_D: ST_CTRL_PID_PARAM;
	rActualValue: REAL;
	FBDCONTROL: FB_D_CONTROL;
	rStFct_CalcZSpeed_D: REAL;
	TONWaitMovement: TON;
	RisingEdgeCountHC: R_TRIG;
	rOutfeedStrokeAxisSpeed: REAL;
	xBlockSetFastVelZAxis: BOOL;
	lrStartRecordMaxTorque: LREAL;
	lrZCheckPosition: LREAL;
	xSetDefaultSpeedS: BOOL;
	lrSaveSSpeed: LREAL;
	xBlockActivateOAxis: BOOL;
	xEndPosReachZylindricalProcess: BOOL;
END_VAR
(****************************************************************************************************************************************************)
(***********                 This Functionblock manage all the station funtion and synchronizing of the Hardware                           ************)
(****************************************************************************************************************************************************)
xActive:=T_Station_Work.TControl.xActiveStation;
IF NOT(T_Station_Work.TControl.xActiveStation) THEN
	IF T_Station_Work.xActive THEN
		T_Station_Work:=TDeleteStationStruct;
	END_IF;
	T_Station_Work.xActive:=FALSE;
	RETURN;
ELSE
	(* Zuweisung der Datenstrukturen der Aktuatoren als Pointer *)
	ptrTAxisZ:=ADR(T_Station_Work.THWWorkStation.TAxisZ);
	ptrTAxisS:=ADR(T_Station_Work.THWWorkStation.TAxisS);
	ptrTCylToolDeflection:=ADR(T_Station_Work.THWWorkStation.TCylToolDeflection);
	ptrTCylToolTorqueHC:=ADR(T_Station_Work.THWWorkStation.TCylToolTorqueHC);
	ptrTCylToolTorqueOverload:=ADR(T_Station_Work.THWWorkStation.TCylToolTorqueOverload);
	ptrTTorqueSensorMeasRange:=ADR(T_Station_Work.THWWorkStation.TTorqueSensorMeasRange);
	ptrTTorqueSensorControl:=ADR(T_Station_Work.THWWorkStation.TTorqueSensorControl);
	ptrTSensorTorque:=ADR(T_Station_Work.THWWorkStation.TSensorTorque);
	ptrTSensorTorqueOverload:=ADR(T_Station_Work.THWWorkStation.TSensorTorqueOverload);
	ptrTCylBrakeReleaseZAxis:=ADR(T_Station_Work.THWWorkStation.TCylBrakeReleaseZAxis);
	ptrTCylWorkpieceClamp:=ADR(T_Station_Work.THWWorkStation.TCylWorkpieceClamp);
	ptrTValveAirTable:=ADR(T_Station_Work.THWWorkStation.TValveAirTable);
	ptrTValveVacuumTable:=ADR(T_Station_Work.THWWorkStation.TValveVacuumTable);
	ptrTValveCleanNozzle:=ADR(T_Station_Work.THWWorkStation.TValveCleanNozzle);
	ptrTAxisBubbler:=ADR(T_Station_Work.THWWorkStation.TAxisBubbler);
	ptrTAxisFeedPump:=ADR(T_Station_Work.THWWorkStation.TAxisFeedPump);
END_IF;
(******************************************************************************************************************************************)
(****************************				                  Status Part                                                            *****************************)
(******************************************************************************************************************************************)
T_Station_Work.xActive:=TRUE;
xStatusRdy:=T_Station_Work.TControl.xRdy;
xStatusEnd:=T_Station_Work.TControl.xDone;
xStatusStop:=xTmpStopFunction;
xStatusRef:=T_Station_Work.TControl.xReferenced;
xError:= T_Station_Work.TControl.xError;
iErrorNr := T_Station_Work.TControl.diErrorNr;
iStatusFctNr:=iStationFunctionNr;
(******************************************************************************************************************************************)
(****************************				                Enable Part                                                            *****************************)
(******************************************************************************************************************************************)
(* Check Active of the Axis Drives *)
xTmp:=	(NOT(ptrTAxisZ^.T_CtrleSingle.xErr) AND NOT(ptrTAxisZ^.T_CtrleSingle.xDone)) OR
		(NOT(ptrTAxisS^.T_CtrleSingle.xErr) AND NOT(ptrTAxisS^.T_CtrleSingle.xDone));
CtrlDisableStation;
CtrlEnableStation;
(******************************************************************************************************************************************)
(****************************				       Security Circuit Switch ON/OFF                                          *****************************)
(******************************************************************************************************************************************)
CtrlSafetySwitch_ON_OFF;
(******************************************************************************************************************************************)
(****************************				         Error Controlling Part                                                  *****************************)
(******************************************************************************************************************************************)
CtrlErrorStation;
(******************************************************************************************************************************************)
(****************************				         Main Controlling Part                                                  *****************************)
(******************************************************************************************************************************************)
CtrlMainStation;
(******************************************************************************************************************************************)
(****************************				            Spindel controlling                                                  *****************************)
(******************************************************************************************************************************************)
StationFunction_Ctrl_ToolSpindle;
(******************************************************************************************************************************************)
(****************************				Überwachung Achsenbremse                                        *****************************)
(******************************************************************************************************************************************)
StationFunction_Ctrl_AxisBrake;
(*****************************************************************************************************************************************)
(****************************				DC Motoren (Suspension)                                        *****************************)
(******************************************************************************************************************************************)
CtrlDCMotors;
(******************************************************************************************************************************************)
(****************************				              Funktionen                                                               *****************************)
(******************************************************************************************************************************************)
xCheckAxisCurrent:=	xSafetyCircuitOn;
IF xStartFunction AND NOT(xSetEnd) AND NOT(xStFct_ForceStationError) THEN
	IF (iStationFunctionNr = 1) THEN
		StationFunction_Fct_01_Referencing;
		T_Station_Work.TControl.wStatus:=wStFct_Status;
	END_IF;
	IF (iStationFunctionNr = 2) THEN
		StationFunction_Fct_02_InitialState;
	END_IF;
	IF (iStationFunctionNr = 3) THEN
		StationFunction_Fct_03_ToolRotationON;
	END_IF;
	IF (iStationFunctionNr = 4) THEN
		StationFunction_Fct_04_InfeedWorking;
		T_Station_Work.TControl.wStatus:=wStFct_Status;
	END_IF;
	IF (iStationFunctionNr = 5) THEN
		StationFunction_Fct_05_Working;
		T_Station_Work.TControl.wStatus:=wStFct_Status;
	END_IF;
	IF (iStationFunctionNr = 6) THEN
		StationFunction_Fct_06_ToolRotationOFF;
	END_IF;
	IF (iStationFunctionNr = 7) THEN
		CASE T_ExchgParam.bToolSpindleActive OF
		1:	(* Maxon Spindel *)
			StationFunction_Fct_07_Calibration;
		2,3:	(* Beckhoff Spindel *)
			StationFunction_Fct_07_Calibration2;
		END_CASE;
	END_IF;
	IF (iStationFunctionNr = 8) THEN
		StationFunction_Fct_08_SpindleBurnIn;
	END_IF;
	IF (iStationFunctionNr = 9) THEN
		StationFunction_Fct_09_Initial_Z_Axis;
	END_IF;
	IF (iStationFunctionNr = 10) THEN
		StationFunction_Fct_10_CheckAxisBreak;
	END_IF;
	IF (iStationFunctionNr = 11) THEN
		StationFunction_Fct_11_Centring;
		T_Station_Work.TControl.wStatus:=wStFct_Status;
	END_IF;
	IF (iStationFunctionNr <> 5) THEN
		T_Z_St1_Ctrle.diVelocityCommandValue:=(T_Z_St1_Ctrle.nOutData2[1] * 65536) + T_Z_St1_Ctrle.nOutData2[0];
		gxZAxisVelocityCtrlActive:=FALSE;
	END_IF;
ELSE
	T_Z_St1_Ctrle.diVelocityCommandValue:=(T_Z_St1_Ctrle.nOutData2[1] * 65536) + T_Z_St1_Ctrle.nOutData2[0];
	gxZAxisVelocityCtrlActive:=FALSE;
END_IF;
(******************************************************************************************************************************************)
(****************************				         Init / Reset Hardware                                                 *****************************)
(******************************************************************************************************************************************)
IF xSetEnd THEN
	xStationError:=FALSE;
	xInitError:=FALSE;
	xInitStart:=FALSE;
	xInitStop:=FALSE;
	xInitStep:=FALSE;
	xSetEnd:=FALSE;
	xTmpStart:=FALSE;
	T_Station_Work.TControl.xExecute:=FALSE;
	T_Station_Work.TControl.xStop:=FALSE;
	T_Station_Work.TControl.xStopCycle:=FALSE;
	T_Station_Work.TControl.xAbord:=FALSE;
	IF NOT(xDontDeleteErrorFlag) THEN
		T_Station_Work.TControl.xDone:=TRUE;
		T_Station_Work.TControl.xError:=FALSE;
		T_Station_Work.TControl.diErrorNr:=0;
	END_IF;
	xDontDeleteErrorFlag:=FALSE;
	xStartFunction:=FALSE;
	xStepError:=FALSE;
	xTmpStationError:=FALSE;
	diErrorNumber:=0;
	xSetError:=FALSE;
	xReadyToQuitErr:=FALSE;
	xStFct_Error:=FALSE;
	T_Station_Work.THWWorkStation.TCtrlWork.xBlockCheckAxisBrake:=FALSE;
END_IF;
IF T_Station_Work.TControl.xRdy THEN
	IF IxJoystick_WorkpieceClamp_ON_St1 THEN
		IF NOT(ptrTCylWorkpieceClamp^.T_CtrleCyl.T_Standard.xActivOn) AND NOT(ptrTCylWorkpieceClamp^.T_CtrleCyl.xExecute) AND ptrTCylWorkpieceClamp^.T_CtrleCyl.xDone THEN
			ptrTCylWorkpieceClamp^.T_CtrleCyl.iFunction:=2;
			ptrTCylWorkpieceClamp^.T_CtrleCyl.xExecute:=TRUE;
		END_IF;
		IF NOT(T_TwinSafeOut.QxContactor24VCh1) OR NOT(T_TwinSafeOut.QxContactor24VCh2) THEN
			T_ExchgParam.T_Visu.T_Message.iState:=230;	(* Warnung: Zuerst die Energieversorgung einschalten ! *)
		END_IF;
	ELSE
		IF ptrTCylWorkpieceClamp^.T_CtrleCyl.T_Standard.xActivOn AND NOT(ptrTCylWorkpieceClamp^.T_CtrleCyl.xExecute) AND ptrTCylWorkpieceClamp^.T_CtrleCyl.xDone THEN
			ptrTCylWorkpieceClamp^.T_CtrleCyl.iFunction:=1;
			ptrTCylWorkpieceClamp^.T_CtrleCyl.xExecute:=TRUE;
		END_IF;
	END_IF;
	IF IxJoystick_AirTable_ON THEN
		IF NOT(ptrTValveAirTable^.T_CtrleCyl.T_Standard.xActivOn) AND NOT(ptrTValveAirTable^.T_CtrleCyl.xExecute) AND ptrTValveAirTable^.T_CtrleCyl.xDone THEN
			ptrTValveAirTable^.T_CtrleCyl.iFunction:=2;
			ptrTValveAirTable^.T_CtrleCyl.xExecute:=TRUE;
		END_IF;
		IF NOT(T_TwinSafeOut.QxContactor24VCh1) OR NOT(T_TwinSafeOut.QxContactor24VCh2) THEN
			T_ExchgParam.T_Visu.T_Message.iState:=230;	(* Warnung: Zuerst die Energieversorgung einschalten ! *)
		END_IF;
	ELSE
		IF ptrTValveAirTable^.T_CtrleCyl.T_Standard.xActivOn AND NOT(ptrTValveAirTable^.T_CtrleCyl.xExecute) AND ptrTValveAirTable^.T_CtrleCyl.xDone THEN
			ptrTValveAirTable^.T_CtrleCyl.iFunction:=1;
			ptrTValveAirTable^.T_CtrleCyl.xExecute:=TRUE;
		END_IF;
	END_IF;
	IF IxJoystick_VaccumTable_ON THEN
		IF NOT(ptrTValveVacuumTable^.T_CtrleCyl.T_Standard.xActivOn) AND NOT(ptrTValveVacuumTable^.T_CtrleCyl.xExecute) AND ptrTValveVacuumTable^.T_CtrleCyl.xDone THEN
			ptrTValveVacuumTable^.T_CtrleCyl.iFunction:=2;
			ptrTValveVacuumTable^.T_CtrleCyl.xExecute:=TRUE;
		END_IF;
		IF NOT(T_TwinSafeOut.QxContactor24VCh1) OR NOT(T_TwinSafeOut.QxContactor24VCh2) THEN
			T_ExchgParam.T_Visu.T_Message.iState:=230;	(* Warnung: Zuerst die Energieversorgung einschalten ! *)
		END_IF;
	ELSE
		IF ptrTValveVacuumTable^.T_CtrleCyl.T_Standard.xActivOn AND NOT(ptrTValveVacuumTable^.T_CtrleCyl.xExecute) AND ptrTValveVacuumTable^.T_CtrleCyl.xDone THEN
			ptrTValveVacuumTable^.T_CtrleCyl.iFunction:=1;
			ptrTValveVacuumTable^.T_CtrleCyl.xExecute:=TRUE;
		END_IF;
	END_IF;
END_IF;

(* Drehmoment Ausgabe *)	(* IGS *)
rStFct_V1:=		T_Station_Parameter.T_OnlineChange.rWorkingSpeedForward;
rStFct_S1:=		0.5;
rStFct_S2:=		T_Station_Parameter.T_OnlineChange.rTorqueLevelHC;
CASE T_ExchgParam.bToolSpindleActive OF
1:	(* Maxon Spindel *)
	rStFct_M:=	T_Station_Parameter.T_TorqueSystem.rActual_Torque;			(* Maxon Spindel ist aktiv *)
	T_ExchgParam.T_StationCommon.rActual_Torque:=T_Station_Parameter.T_TorqueSystem.rActual_Torque;	(* für MMI *)
	T_ExchgParam.T_StationCommon.rMaxTorque:=T_Station_Parameter.T_TorqueSystem.rMaxTorque;			(* für MMI *)
2:	(* Beckhoff Spindel L *)
	rStFct_M:=	T_Station_Parameter.T_TorqueSystem_L.rActual_Torque;		(* Beckhoff Spindel ist aktiv *)
	T_ExchgParam.T_StationCommon.rActual_Torque:=T_Station_Parameter.T_TorqueSystem_L.rActual_Torque;	(* für MMI *)
	T_ExchgParam.T_StationCommon.rMaxTorque:=T_Station_Parameter.T_TorqueSystem_L.rMaxTorque;		(* für MMI *)
3:	(* Beckhoff Spindel M *)
	rStFct_M:=	T_Station_Parameter.T_TorqueSystem_M.rActual_Torque;		(* Beckhoff Spindel ist aktiv *)
	T_ExchgParam.T_StationCommon.rActual_Torque:=T_Station_Parameter.T_TorqueSystem_M.rActual_Torque;	(* für MMI *)
	T_ExchgParam.T_StationCommon.rMaxTorque:=T_Station_Parameter.T_TorqueSystem_M.rMaxTorque;		(* für MMI *)
END_CASE;
IF NOT(xStartFunction) THEN
	(* Regelung mit Override Funktion und mit Parabelfunktion und mit prozentualer Angabe der Regelungssteigung mit oder ohne konstante Geschwindigkeit *)
	T_Station_Work.THWWorkStation.TCtrlWork.rSpeedZ_V1:=rStFct_V1;
	T_Station_Work.THWWorkStation.TCtrlWork.rTorqueZ_S4:=rStFct_S2;
END_IF;
T_Station_Work.THWWorkStation.TCtrlWork.rSpeedZ_V3:=rStFct_V1/100.0;
T_Station_Work.THWWorkStation.TCtrlWork.rTorqueZ_S1:=rStFct_S1;
T_Station_Work.THWWorkStation.TCtrlWork.rTorqueHC:=rStFct_S2;
T_Station_Parameter.T_InfoProcess.rTorqueHC:=T_Station_Work.THWWorkStation.TCtrlWork.rTorqueHC;
(***************************************************************************************************************************************************)
(* Ausgabe Drehmoment für Progressbalken *)
IF (T_Station_Work.THWWorkStation.TCtrlWork.rTorqueHC <> 0.0) THEN
	T_Station_Work.THWWorkStation.TCtrlWork.iProgressBar_Torque:=REAL_TO_INT(100.0/T_Station_Work.THWWorkStation.TCtrlWork.rTorqueHC*rStFct_M);
ELSE
	T_Station_Work.THWWorkStation.TCtrlWork.iProgressBar_Torque:=0;
END_IF;
IF (T_Station_Work.THWWorkStation.TCtrlWork.iProgressBar_Torque < 0) THEN
	T_Station_Work.THWWorkStation.TCtrlWork.iProgressBar_Torque:=0;
END_IF;
(***************************************************************************************************************************************************)
(* Ausgabe Z Position und Geschwindigkeit für Progressbalken *)

